// TwinCAT 3 PLC project mobject_collections
// Title: mobject-collections
// Company: mobject
// Author: mobject dev team
// ProjectVersion: 1.3.0
// ProgramVersion: 3.1.4023.0
// libraries:
//   Tc2_System, * (Beckhoff Automation GmbH)
//   Tc3_DynamicMemory, * (Beckhoff Automation GmbH)
//   mobject-disposable,1.1.1,mobject
//   mobject-enumerable,1.2.0,mobject
//   mobject-events,1.1.0,mobject
// project tree:
//   Dictionary/ Dictionary.TcPOU
//   Interfaces/Collections/Events/ I_CollectionChangedEvent.TcIO, I_CollectionDisposedEvent.TcIO (not stored)
//   Interfaces/Collections/ I_Collection.TcIO, I_List.TcIO, I_LinkedList.TcIO, I_Queue.TcIO, I_Stack.TcIO
//   Interfaces/Collections/Nodes/ I_CollectionNode.TcIO, I_LinkedListNode.TcIO, I_ListNode.TcIO
//   Interfaces/KeyValueCollections/Events/ I_KeyValueCollectionChangedEvent.TcIO, I_KeyValueCollectionDisposedEvent.TcIO
//   Interfaces/KeyValueCollections/ I_Dictionary.TcIO, I_KeyValueCollection.TcIO
//   Interfaces/KeyValueCollections/Nodes/ I_DictionaryTreeNode.TcIO, I_OrderedDictionaryTreeNode.TcIO
//   LinkedList/ LinkedList.TcPOU
//   List/ List.TcPOU
//   OrderedDictionary/ OrderedDictionary.TcPOU
//   Queue/ Queue.TcPOU
//   Stack/ Stack.TcPOU
//   _Internal/Dictionary/Enumerator/ DictionaryForwardEnumerator.TcPOU
//   _Internal/Dictionary/Node/ DictionaryTreeNode.TcPOU
//   _Internal/Events/Collection/ CollectionChangedEvent.TcPOU, CollectionDisposedEvent.TcPOU, CollectionEvent.TcPOU
//   _Internal/Events/KeyValueCollection/ KeyValueCollectionChangedEvent.TcPOU, KeyValueCollectionDisposedEvent.TcPOU, KeyValueCollectionEvent.TcPOU
//   _Internal/LinkedList/Enumerator/ LinkedListForwardEnumerator.TcPOU
//   _Internal/LinkedList/Node/ LinkedListNode.TcPOU
//   _Internal/List/Enumerator/ ListForwardEnumerator.TcPOU
//   _Internal/List/Node/ ListNode.TcPOU
//   _Internal/OrderedDictionary/Enumerator/ OrderedDictionaryForwardEnumerator.TcPOU
//   _Internal/OrderedDictionary/Node/ OrderedDictionaryTreeNode.TcPOU

// ---- Interfaces/Collections/Events/I_CollectionChangedEvent.TcIO
INTERFACE I_CollectionChangedEvent EXTENDS I_Event

PROPERTY PUBLIC Target : I_Collection
GET
END_GET
END_PROPERTY

END_INTERFACE

// ---- Interfaces/Collections/I_Collection.TcIO
INTERFACE I_Collection EXTENDS I_Enumerable, I_Disposable, I_EventEmitter

METHOD PUBLIC AddItem
VAR_INPUT
	Item : ANY;
END_VAR
END_METHOD

METHOD PUBLIC Clear
END_METHOD

METHOD PUBLIC Contains : BOOL;
VAR_INPUT
	Item : ANY;
END_VAR
END_METHOD

PROPERTY PUBLIC Count : DINT
GET
END_GET
END_PROPERTY

PROPERTY IsEmpty : BOOL
GET
END_GET
END_PROPERTY

METHOD PUBLIC TryCopyTo : BOOL
VAR_INPUT
	Destination : ANY;
END_VAR
END_METHOD

METHOD PUBLIC TryCopyToLocation : BOOL
VAR_INPUT
	DestinationAddress : PVOID;
	DestinationSize : UDINT;
END_VAR
END_METHOD

METHOD PUBLIC TryRemoveItem : BOOL
VAR_INPUT
	Item : ANY;
END_VAR
END_METHOD

END_INTERFACE

// ---- Interfaces/Collections/I_List.TcIO
INTERFACE I_List EXTENDS I_Collection

PROPERTY PUBLIC Capacity : DINT
GET
END_GET
END_PROPERTY

METHOD PUBLIC GetIndexOf : DINT
VAR_INPUT
	Item : ANY;
END_VAR
END_METHOD

METHOD PUBLIC TrimExcess
END_METHOD

METHOD PUBLIC TryGetByIndex : BOOL
VAR_INPUT
	Index : DINT;
	Destination : ANY;
END_VAR
END_METHOD

METHOD PUBLIC TryGetToByIndex : BOOL
VAR_INPUT
	Index : DINT;
	DestinationAddress : PVOID;
	DestinationSize : UDINT;
END_VAR
END_METHOD

METHOD TryInsert : BOOL
VAR_INPUT
	Index : DINT;
	Item : ANY;
END_VAR
END_METHOD

METHOD TryRemoveAt : BOOL
VAR_INPUT
	Index : DINT;
END_VAR
END_METHOD

END_INTERFACE

// ---- Interfaces/Collections/I_LinkedList.TcIO
INTERFACE I_LinkedList EXTENDS I_Collection

METHOD PUBLIC AddAfter
VAR_INPUT
	After : I_LinkedListNode;
	Value : ANY;
END_VAR
END_METHOD

METHOD PUBLIC AddBefore
VAR_INPUT
	Before : I_LinkedListNode;
	Value : ANY;
END_VAR
END_METHOD

METHOD PUBLIC AddFirst
VAR_INPUT
	Value : ANY;
END_VAR
END_METHOD

METHOD PUBLIC AddLast
VAR_INPUT
	Value : ANY;
END_VAR
END_METHOD

METHOD PUBLIC Find : I_LinkedListNode
VAR_INPUT
	Value : ANY;
END_VAR
END_METHOD

METHOD PUBLIC FindLast : I_LinkedListNode
VAR_INPUT
	Value : ANY;
END_VAR
END_METHOD

PROPERTY PUBLIC First : I_LinkedListNode
GET
END_GET
END_PROPERTY

PROPERTY PUBLIC Last : I_LinkedListNode
GET
END_GET
END_PROPERTY

METHOD PUBLIC Remove
VAR_INPUT
	Value : ANY;
END_VAR
END_METHOD

METHOD PUBLIC RemoveFirst
END_METHOD

METHOD PUBLIC RemoveLast
END_METHOD

END_INTERFACE

// ---- Interfaces/Collections/I_Queue.TcIO
INTERFACE I_Queue EXTENDS I_Collection

METHOD PUBLIC Enqueue
VAR_INPUT
	Item : ANY;
END_VAR
END_METHOD

METHOD PUBLIC TryDequeue : BOOL;
VAR_INPUT
	Destination : ANY;
END_VAR
END_METHOD

METHOD PUBLIC TryPeek : BOOL;
VAR_INPUT
	Destination : ANY;
END_VAR
END_METHOD

END_INTERFACE

// ---- Interfaces/Collections/I_Stack.TcIO
INTERFACE I_Stack EXTENDS I_Collection, I_EventEmitter

METHOD PUBLIC Push
VAR_INPUT
	Item : ANY;
END_VAR
END_METHOD

METHOD PUBLIC TryPeek : BOOL;
VAR_INPUT
	Destination : ANY;
END_VAR
END_METHOD

METHOD PUBLIC TryPop : BOOL;
VAR_INPUT
	Destination : ANY;
END_VAR
END_METHOD

END_INTERFACE

// ---- Interfaces/Collections/Nodes/I_CollectionNode.TcIO
INTERFACE I_CollectionNode EXTENDS I_Disposable

PROPERTY PUBLIC DataSize : UDINT
GET
END_GET
END_PROPERTY

METHOD PUBLIC Equals : BOOL
VAR_INPUT
	Symbol : ANY;
END_VAR
END_METHOD

METHOD PUBLIC TryGet : BOOL;
VAR_INPUT
	Destination : ANY;
END_VAR
END_METHOD

METHOD PUBLIC TryGetTo : BOOL;
VAR_INPUT
	DestinationAddress : PVOID;
	DestinationSize : UDINT;
END_VAR
END_METHOD

END_INTERFACE

// ---- Interfaces/Collections/Nodes/I_LinkedListNode.TcIO
INTERFACE I_LinkedListNode EXTENDS I_CollectionNode

PROPERTY PUBLIC Next : I_LinkedListNode
GET
END_GET
SET
END_SET
END_PROPERTY

PROPERTY PUBLIC Previous : I_LinkedListNode
GET
END_GET
SET
END_SET
END_PROPERTY

END_INTERFACE

// ---- Interfaces/Collections/Nodes/I_ListNode.TcIO
INTERFACE I_ListNode EXTENDS I_CollectionNode;

END_INTERFACE

// ---- Interfaces/KeyValueCollections/Events/I_KeyValueCollectionChangedEvent.TcIO
INTERFACE I_KeyValueCollectionChangedEvent EXTENDS I_Event

PROPERTY PUBLIC Target : I_KeyValueCollection
GET
END_GET
END_PROPERTY

END_INTERFACE

// ---- Interfaces/KeyValueCollections/Events/I_KeyValueCollectionDisposedEvent.TcIO
INTERFACE I_KeyValueCollectionDisposedEvent EXTENDS I_Event

PROPERTY PUBLIC Target : I_KeyValueCollection
GET
END_GET
END_PROPERTY

END_INTERFACE

// ---- Interfaces/KeyValueCollections/I_Dictionary.TcIO
INTERFACE I_Dictionary EXTENDS I_KeyValueCollection

METHOD PUBLIC AddOrUpdate
VAR_INPUT
	Key : T_MAXSTRING;
	Value : ANY;
END_VAR
END_METHOD

METHOD PUBLIC Clear
VAR_INPUT
END_VAR
END_METHOD

METHOD PUBLIC ContainsKey : BOOL
VAR_INPUT
	Key : T_MAXSTRING;
END_VAR
END_METHOD

METHOD PUBLIC GetKeys : I_Collection
END_METHOD

PROPERTY IsEmpty : BOOL
GET
END_GET
END_PROPERTY

METHOD PUBLIC Remove
VAR_INPUT
	Key : T_MAXSTRING;
END_VAR
END_METHOD

METHOD PUBLIC TryAdd : BOOL
VAR_INPUT
	Key : T_MAXSTRING;
	Value : ANY;
END_VAR
END_METHOD

METHOD PUBLIC TryGetValue : BOOL
VAR_INPUT
	Key : T_MAXSTRING;
	Destination	: ANY;
END_VAR
END_METHOD

METHOD PUBLIC TryGetValueTo : BOOL
VAR_INPUT
	Key : T_MAXSTRING;
	DestinationAddress : PVOID;
	DestinationSize : UDINT;
END_VAR
END_METHOD

END_INTERFACE

// ---- Interfaces/KeyValueCollections/I_KeyValueCollection.TcIO
INTERFACE I_KeyValueCollection EXTENDS I_KeyValueEnumerable, I_Enumerable, I_Disposable, I_EventEmitter

END_INTERFACE

// ---- Interfaces/KeyValueCollections/Nodes/I_DictionaryTreeNode.TcIO
INTERFACE I_DictionaryTreeNode EXTENDS I_CollectionNode

METHOD PUBLIC Clone
VAR_INPUT
	Node : I_DictionaryTreeNode;
END_VAR
END_METHOD

PROPERTY PUBLIC Height : DINT
GET
END_GET
SET
END_SET
END_PROPERTY

PROPERTY PUBLIC Key : T_MAXSTRING
GET
END_GET
END_PROPERTY

PROPERTY PUBLIC Left : I_DictionaryTreeNode
GET
END_GET
SET
END_SET
END_PROPERTY

PROPERTY PUBLIC NodeBufferPointer : Pointer To Byte
GET
END_GET
END_PROPERTY

PROPERTY PUBLIC NodeBufferSize : UDINT
GET
END_GET
END_PROPERTY

METHOD Reinitialize
VAR_INPUT
	Key : T_MAXSTRING;
	Source : ANY;
END_VAR
END_METHOD

PROPERTY PUBLIC Right : I_DictionaryTreeNode
GET
END_GET
SET
END_SET
END_PROPERTY

END_INTERFACE

// ---- Interfaces/KeyValueCollections/Nodes/I_OrderedDictionaryTreeNode.TcIO
INTERFACE I_OrderedDictionaryTreeNode EXTENDS I_CollectionNode

METHOD PUBLIC Clone
VAR_INPUT
	Node : I_OrderedDictionaryTreeNode;
END_VAR
END_METHOD

PROPERTY PUBLIC Height : DINT
GET
END_GET
SET
END_SET
END_PROPERTY

PROPERTY PUBLIC Key : T_MAXSTRING
GET
END_GET
END_PROPERTY

PROPERTY PUBLIC Left : I_OrderedDictionaryTreeNode
GET
END_GET
SET
END_SET
END_PROPERTY

PROPERTY PUBLIC Next : I_OrderedDictionaryTreeNode
GET
END_GET
SET
END_SET
END_PROPERTY

PROPERTY PUBLIC NodeBufferPointer : Pointer To Byte
GET
END_GET
END_PROPERTY

PROPERTY PUBLIC NodeBufferSize : UDINT
GET
END_GET
END_PROPERTY

PROPERTY PUBLIC Previous : I_OrderedDictionaryTreeNode
GET
END_GET
SET
END_SET
END_PROPERTY

METHOD Reinitialize
VAR_INPUT
	Key : T_MAXSTRING;
	Source : ANY;
END_VAR
END_METHOD

PROPERTY PUBLIC Right : I_OrderedDictionaryTreeNode
GET
END_GET
SET
END_SET
END_PROPERTY

END_INTERFACE

// ---- Dictionary/Dictionary.TcPOU
{attribute 'linkalways'} 
{attribute 'no_explicit_call' := 'This FB is a CLASS and must be accessed using methods or properties'}
{attribute 'enable_dynamic_creation'}
FUNCTION_BLOCK Dictionary EXTENDS Disposable IMPLEMENTS I_Dictionary
VAR
	eventEmitter : EventEmitter;
	rootNode : I_DictionaryTreeNode;
END_VAR

METHOD PUBLIC AddOrUpdate
VAR_INPUT
	Key : T_MAXSTRING;
	Value : ANY;
END_VAR
rootNode := THIS^.RecursiveInsert(Key, Value, rootNode);
EmitChangedEvent();
END_METHOD

METHOD PRIVATE Balance : I_DictionaryTreeNode
VAR_INPUT
	Node : I_DictionaryTreeNode;
END_VAR
VAR
	balanceFactor : DINT;
END_VAR
balanceFactor := THIS^.GetBalanceFactor(Node);

IF (balanceFactor > 1) THEN
	IF THIS^.GetBalanceFactor(Node.Left) < 0 THEN
		Node.Left := THIS^.LeftRotate(Node.Left);
	END_IF
	Node := RightRotate(Node);
ELSIF (balanceFactor < -1) THEN
	IF THIS^.GetBalanceFactor(Node.Right) > 0 THEN
		Node.Right := RightRotate(Node.Right);
	END_IF
	Node := LeftRotate(Node);
END_IF

Balance := Node;
END_METHOD

METHOD PUBLIC Clear
VAR_INPUT
END_VAR
IF rootNode = 0 THEN
	RETURN;
END_IF

THIS^.RecursiveClear(rootNode);
rootNode := 0;
EmitChangedEvent();
END_METHOD

METHOD PUBLIC ContainsKey : BOOL
VAR_INPUT
	Key : T_MAXSTRING;
END_VAR
VAR
	foundNode : I_DictionaryTreeNode;
END_VAR
foundNode := THIS^.RecursiveFind(Key, rootNode);

IF foundNode = 0 THEN
	RETURN;
END_IF

ContainsKey := TRUE;
END_METHOD

PROPERTY PUBLIC Count : DINT
GET
VAR
	NodeCount : DINT;
END_VAR
RecursiveCountNodes(rootNode, NodeCount);
Count := NodeCount;
END_GET
END_PROPERTY

METHOD PRIVATE EmitChangedEvent
VAR
	pDictionaryChangedEvent : POINTER TO KeyValueCollectionChangedEvent;
END_VAR
pDictionaryChangedEvent := __NEW(KeyValueCollectionChangedEvent(Target := THIS^));
eventEmitter.Emit('OnChanged', pDictionaryChangedEvent^);
pDictionaryChangedEvent^.Dispose();
END_METHOD

METHOD PRIVATE EmitDisposedEvent
VAR
	pDictionaryDisposedEvent : POINTER TO KeyValueCollectionDisposedEvent;
END_VAR
pDictionaryDisposedEvent := __NEW(KeyValueCollectionDisposedEvent(Target := THIS^));
eventEmitter.Emit('OnDisposed', pDictionaryDisposedEvent^);
pDictionaryDisposedEvent^.Dispose();
END_METHOD

METHOD FB_exit : BOOL
VAR_INPUT
	bInCopyCode : BOOL; // if TRUE, the exit method is called for exiting an instance that is copied afterwards (online change).
END_VAR
VAR
END_VAR
IF bInCopyCode THEN
    RETURN;
END_IF

Clear();
EmitDisposedEvent();
END_METHOD

METHOD PRIVATE FindMinimum : I_DictionaryTreeNode
VAR_INPUT
	Node : I_DictionaryTreeNode;
END_VAR
VAR
	nextNode : I_DictionaryTreeNode;
END_VAR
nextNode := Node;

WHILE (nextNode.left <> 0) DO
      nextNode := nextNode.left;
END_WHILE;

FindMinimum := nextNode;
END_METHOD

METHOD PRIVATE GetBalanceFactor : DINT
VAR_INPUT
	Node : I_DictionaryTreeNode;
END_VAR
IF (Node = 0) THEN
	GetBalanceFactor := 0;
	RETURN;
END_IF

GetBalanceFactor := THIS^.GetHeight(node.left) - THIS^.GetHeight(node.right);
END_METHOD

METHOD GetEnumerator : I_ForwardEnumerator
VAR
	pNodeCollection : POINTER TO LinkedList;
	pEnumerator : POINTER TO DictionaryForwardEnumerator;
END_VAR
pNodeCollection := __NEW(LinkedList);
THIS^.RecursiveAddNodesInOrderToCollection(rootNode, pNodeCollection^);

pEnumerator := __NEW(DictionaryForwardEnumerator(Parent := THIS^, Nodes := pNodeCollection^));
GetEnumerator := pEnumerator^;
END_METHOD

METHOD PRIVATE GetHeight : DINT
VAR_INPUT
	Node : I_DictionaryTreeNode;
END_VAR
IF Node = 0 THEN
	GetHeight := -1;
	RETURN;
END_IF

GetHeight := Node.Height;
END_METHOD

METHOD PUBLIC GetKeys : I_Collection
VAR
	pLinkedList : POINTER TO LinkedList;
END_VAR
pLinkedList := __NEW(LinkedList);
THIS^.RecursiveAddKeysInOrderToCollection(rootNode,pLinkedList^);
GetKeys := pLinkedList^;
END_METHOD

METHOD GetKeyValueEnumerator : I_KeyValueForwardEnumerator
VAR
	pNodeCollection : POINTER TO LinkedList;
	pEnumerator : POINTER TO DictionaryForwardEnumerator;
END_VAR
pNodeCollection := __NEW(LinkedList);
THIS^.RecursiveAddNodesInOrderToCollection(rootNode, pNodeCollection^);

pEnumerator := __NEW(DictionaryForwardEnumerator(Parent := THIS^, Nodes := pNodeCollection^));
GetKeyValueEnumerator := pEnumerator^;
END_METHOD

METHOD PRIVATE LeftRotate : I_DictionaryTreeNode
VAR_INPUT
	X : I_DictionaryTreeNode;
END_VAR
VAR
	y : I_DictionaryTreeNode;
	t2 : I_DictionaryTreeNode;
END_VAR
y := X.right;
t2 := y.left;
y.left := X;
X.right := t2;
THIS^.UpdateHeight(X);
THIS^.UpdateHeight(y);
LeftRotate := y;
END_METHOD

METHOD PUBLIC OffEvent
VAR_INPUT
	EventName : T_MaxString;
	EventHandler : I_EventHandler;
END_VAR
eventEmitter.OffEvent(EventName, EventHandler);
END_METHOD

METHOD PUBLIC OnceEvent
VAR_INPUT
	EventName : T_MaxString;
	EventHandler : I_EventHandler;
END_VAR
eventEmitter.OnceEvent(EventName, EventHandler);
END_METHOD

METHOD PUBLIC OnEvent
VAR_INPUT
	EventName : T_MaxString;
	EventHandler : I_EventHandler;
END_VAR
eventEmitter.OnEvent(EventName, EventHandler);
END_METHOD

METHOD PRIVATE RecursiveAddKeysInOrderToCollection
VAR_INPUT
	Node : I_DictionaryTreeNode;
	Collection : I_Collection;
END_VAR
VAR
	key : T_MAXSTRING;
END_VAR
IF Node = 0 THEN
	RETURN;
END_IF

THIS^.RecursiveAddKeysInOrderToCollection(Node.Left,Collection);
key := Node.Key;
Collection.AddItem(key);
THIS^.RecursiveAddKeysInOrderToCollection(Node.Right,Collection);
END_METHOD

METHOD PRIVATE RecursiveAddNodesInOrderToCollection
VAR_INPUT
	Node : I_DictionaryTreeNode;
	Collection : I_Collection;
END_VAR
IF Node = 0 THEN
	RETURN;
END_IF

THIS^.RecursiveAddNodesInOrderToCollection(Node.Left,Collection);
Collection.AddItem(Node);
THIS^.RecursiveAddNodesInOrderToCollection(Node.Right,Collection);
END_METHOD

METHOD PRIVATE RecursiveClear
VAR_INPUT
	Node : I_DictionaryTreeNode;
END_VAR
VAR
	thisNodeKey : T_MAXSTRING;
	leftNodeKey : T_MAXSTRING;
	rightNodeKey : T_MAXSTRING;
END_VAR
IF (Node = 0) THEN
	RETURN;
END_IF

thisNodeKey := Node.key;

IF (Node.Left <> 0) THEN
	leftNodeKey := Node.Left.key;
END_IF

IF (Node.Right <> 0) THEN
	rightNodeKey := Node.Right.key;
END_IF


RecursiveClear(Node.Left);
RecursiveClear(Node.Right);
Node.Dispose();
END_METHOD

METHOD PRIVATE RecursiveCountNodes
VAR_INPUT
	Node : I_DictionaryTreeNode;
	Count : REFERENCE TO DINT;
END_VAR
IF Node = 0 THEN
	RETURN;
END_IF

Count := Count + 1;

THIS^.RecursiveCountNodes(Node.Left,Count);
THIS^.RecursiveCountNodes(Node.Right,Count);
END_METHOD

METHOD PRIVATE RecursiveDelete : I_DictionaryTreeNode
VAR_INPUT
	Key : T_MAXSTRING;
	Node : I_DictionaryTreeNode;
END_VAR
VAR
	newNode : I_DictionaryTreeNode; 
	minValueNode : I_DictionaryTreeNode;
	minValueNodeParent : I_DictionaryTreeNode;
	balanceFactor : DINT;
END_VAR
IF (Node = 0) THEN
    RETURN;
END_IF

IF (Key < Node.Key) THEN
    Node.left := THIS^.RecursiveDelete(Key, Node.left);
ELSIF (Key > Node.Key) THEN
    Node.right := THIS^.RecursiveDelete(Key, Node.right);
ELSE
    IF (Node.Left = 0) OR (Node.Right = 0) THEN
        IF (Node.Left = 0) THEN
            newNode := Node.Right;
        ELSE
            newNode := Node.Left;
        END_IF

        Node.Dispose();
        THIS^.updateHeight(newNode);
        RecursiveDelete := THIS^.Balance(newNode);
        RETURN;
    ELSE
        minValueNode := FindMinimum(Node.Right);
        Node.Clone(minValueNode);
        Node.Right := THIS^.RecursiveDelete(minValueNode.Key, Node.Right);	
    END_IF
END_IF

THIS^.updateHeight(Node);
RecursiveDelete := THIS^.Balance(Node);
END_METHOD

METHOD PRIVATE RecursiveFind : I_DictionaryTreeNode
VAR_INPUT
	Key : T_MAXSTRING;
	Node : I_DictionaryTreeNode;
END_VAR
IF (Node = 0) THEN
	RETURN;
END_IF

IF (Key < Node.key) THEN
  RecursiveFind := THIS^.RecursiveFind(key, Node.left);
  RETURN;
ELSIF (key > Node.key) THEN
  RecursiveFind := THIS^.RecursiveFind(key, Node.right);
  RETURN;
ELSE 
  RecursiveFind := Node;
  RETURN;
END_IF
END_METHOD

METHOD PRIVATE RecursiveInsert : I_DictionaryTreeNode
VAR_INPUT
	Key : T_MAXSTRING;
	Value : ANY;
	Node : I_DictionaryTreeNode;
END_VAR
VAR
	pAVLTreeNode : POINTER TO DictionaryTreeNode;
	balanceFactor : DINT;
END_VAR
IF (Node = 0) THEN
	pAVLTreeNode := __NEW(DictionaryTreeNode(NodeKey := Key, NodeSource := Value));
	RecursiveInsert := pAVLTreeNode^;
	RETURN;
END_IF

IF (Key < Node.Key) THEN
	Node.left := THIS^.RecursiveInsert(Key, Value, Node.left);
ELSIF (Key > Node.Key) THEN
	Node.right := THIS^.RecursiveInsert(Key, Value, Node.right);
ELSE
	Node.Reinitialize(Key,Value);
	RecursiveInsert := Node;
END_IF

THIS^.updateHeight(node);

balanceFactor := THIS^.GetBalanceFactor(Node);
Node := balance(Node);
RecursiveInsert := Node;
END_METHOD

METHOD PUBLIC Remove
VAR_INPUT
	Key : T_MAXSTRING;
END_VAR
rootNode := THIS^.RecursiveDelete(Key, rootNode);
EmitChangedEvent();
END_METHOD

METHOD PRIVATE RightRotate : I_DictionaryTreeNode
VAR_INPUT
	Y : I_DictionaryTreeNode;
END_VAR
VAR
	x : I_DictionaryTreeNode;
	t2 : I_DictionaryTreeNode;
END_VAR
x := Y.left;
t2 := x.right;
x.right := Y;
Y.left := t2;
THIS^.UpdateHeight(Y);
THIS^.UpdateHeight(x);
RightRotate := x;
END_METHOD

METHOD PUBLIC TryAdd : BOOL
VAR_INPUT
	Key : T_MAXSTRING;
	Value : ANY;
END_VAR
IF ContainsKey(Key) THEN
	RETURN;
END_IF
	  
THIS^.AddOrUpdate(Key, Value);
TryAdd := TRUE;
END_METHOD

METHOD PUBLIC TryGetValue : BOOL
VAR_INPUT
	Key : T_MAXSTRING;
	Destination	: ANY;
END_VAR
TryGetValue := TryGetValueTo(Key, Destination.pValue, DINT_TO_UDINT(Destination.diSize));
END_METHOD

METHOD PUBLIC TryGetValueTo : BOOL
VAR_INPUT
	Key : T_MAXSTRING;
	DestinationAddress : PVOID;
	DestinationSize : UDINT;
END_VAR
VAR
	foundNode : I_DictionaryTreeNode;
END_VAR
foundNode := THIS^.RecursiveFind(Key, rootNode);

IF foundNode = 0 THEN
	RETURN;
END_IF

TryGetValueTo := foundNode.TryGetTo(DestinationAddress, DestinationSize);
END_METHOD

METHOD PRIVATE UpdateHeight
VAR_INPUT
	Node : I_DictionaryTreeNode;
END_VAR
IF (Node = 0) THEN
	RETURN;
END_IF

Node.height := 1 + MAX(THIS^.GetHeight(Node.left), THIS^.GetHeight(Node.right));
END_METHOD

END_FUNCTION_BLOCK

// ---- _Internal/Events/KeyValueCollection/KeyValueCollectionChangedEvent.TcPOU
{attribute 'linkalways'} 
{attribute 'no_explicit_call' := 'This FB is a CLASS and must be accessed using methods or properties'}
{attribute 'enable_dynamic_creation'}
FUNCTION_BLOCK KeyValueCollectionChangedEvent EXTENDS KeyValueCollectionEvent IMPLEMENTS I_KeyValueCollectionChangedEvent

END_FUNCTION_BLOCK

// ---- _Internal/Events/KeyValueCollection/KeyValueCollectionEvent.TcPOU
{attribute 'linkalways'} 
{attribute 'no_explicit_call' := 'This FB is a CLASS and must be accessed using methods or properties'}
{attribute 'enable_dynamic_creation'}
FUNCTION_BLOCK ABSTRACT KeyValueCollectionEvent EXTENDS Disposable
VAR
	_target : I_KeyValueCollection;
END_VAR

METHOD FB_init : BOOL
VAR_INPUT
	bInitRetains : BOOL; // if TRUE, the retain variables are initialized (warm start / cold start)
	bInCopyCode : BOOL;  // if TRUE, the instance afterwards gets moved into the copy code (online change)
	Target : I_KeyValueCollection;
END_VAR
This^._target := Target;
END_METHOD

PROPERTY PUBLIC Target : I_KeyValueCollection
GET // PUBLIC
Target := _target;
END_GET
END_PROPERTY

END_FUNCTION_BLOCK

// ---- _Internal/Events/KeyValueCollection/KeyValueCollectionDisposedEvent.TcPOU
{attribute 'linkalways'} 
{attribute 'no_explicit_call' := 'This FB is a CLASS and must be accessed using methods or properties'}
{attribute 'enable_dynamic_creation'}
FUNCTION_BLOCK KeyValueCollectionDisposedEvent EXTENDS KeyValueCollectionEvent IMPLEMENTS I_KeyValueCollectionDisposedEvent

END_FUNCTION_BLOCK

// ---- LinkedList/LinkedList.TcPOU
{attribute 'linkalways'} 
{attribute 'no_explicit_call' := 'This FB is a CLASS and must be accessed using methods or properties'}
{attribute 'enable_dynamic_creation'}
FUNCTION_BLOCK LinkedList EXTENDS Disposable IMPLEMENTS I_LinkedList
VAR
	head : I_LinkedListNode;
	tail : I_LinkedListNode;
	eventEmitter : EventEmitter;
END_VAR

METHOD PUBLIC AddAfter
VAR_INPUT
	After : I_LinkedListNode;
	Value : ANY;
END_VAR
VAR
	node : I_LinkedListNode;
END_VAR
IF NOT ContainsLinkedListNode(After) THEN
	RETURN;
END_IF

node := CreateNode(Value);
AddNodeAfter(After,node);
EmitChangedEvent();
END_METHOD

METHOD PUBLIC AddBefore
VAR_INPUT
	Before : I_LinkedListNode;
	Value : ANY;
END_VAR
VAR
	node : I_LinkedListNode;
END_VAR
IF NOT ContainsLinkedListNode(Before) THEN
	RETURN;
END_IF

node := CreateNode(Value);
AddNodeBefore(Before,node);
EmitChangedEvent();
END_METHOD

METHOD PUBLIC AddFirst
VAR_INPUT
	Value : ANY;
END_VAR
VAR
	node : I_LinkedListNode;
END_VAR
node := CreateNode(Value);
AddNodeFirst(node);
EmitChangedEvent();
END_METHOD

METHOD PUBLIC AddItem
VAR_INPUT
	Item : ANY;
END_VAR
AddLast(Item);
END_METHOD

METHOD PUBLIC AddLast
VAR_INPUT
	Value : ANY;
END_VAR
VAR
	node : I_LinkedListNode;
END_VAR
node := CreateNode(Value);
AddNodeLast(node);
EmitChangedEvent();
END_METHOD

METHOD PRIVATE AddNodeAfter
VAR_INPUT
	After : I_LinkedListNode;
	Node : I_LinkedListNode;
END_VAR
VAR
	originalNext : I_LinkedListNode;
END_VAR
IF After = tail THEN
	AddNodeLast(Node);
	RETURN;
END_IF

originalNext := After.Next;
After.Next := Node;
Node.Previous := After;
Node.Next := originalNext;
originalNext.Previous := Node;
END_METHOD

METHOD PRIVATE AddNodeBefore
VAR_INPUT
	Before : I_LinkedListNode;
	Node : I_LinkedListNode;
END_VAR
VAR
	originalBefore : I_LinkedListNode;
END_VAR
IF Before = head THEN
	AddNodeFirst(Node);
	RETURN;
END_IF

originalBefore := Before.Previous;
Before.Previous := Node;
Node.Next := Before;
Node.Previous := originalBefore;
originalBefore.Next := Node;
END_METHOD

METHOD PRIVATE AddNodeFirst
VAR_INPUT
	Node : I_LinkedListNode;
END_VAR
VAR
	originalFirst : I_LinkedListNode;
END_VAR
IF IsEmpty THEN
	head := Node;
	tail := Node; 
	RETURN;	
END_IF

originalFirst := head;
head := Node;
Node.Next := originalFirst;
originalFirst.Previous := Node;
END_METHOD

METHOD PRIVATE AddNodeLast
VAR_INPUT
	Node : I_LinkedListNode;
END_VAR
VAR
	originalLast : I_LinkedListNode;
END_VAR
IF IsEmpty THEN
	head := Node;
	tail := Node; 
	RETURN;	
END_IF

originalLast := tail;
tail := Node;
Node.Previous := originalLast;
originalLast.Next := Node;
END_METHOD

METHOD PUBLIC Clear
IF IsEmpty THEN
	return;
END_IF

RemoveAllNodes();
EmitChangedEvent();
END_METHOD

METHOD PUBLIC Contains : BOOL
VAR_INPUT
    Item : ANY;
END_VAR
VAR
    found : I_LinkedListNode;
END_VAR
found := Find(Item);
Contains := found <> 0;
END_METHOD

METHOD PRIVATE ContainsLinkedListNode : BOOL
VAR_INPUT
    Node : I_LinkedListNode;
END_VAR
VAR
	current : I_LinkedListNode;
END_VAR
IF IsEmpty THEN	
	RETURN;
END_IF

current := head; 

WHILE current <> 0 DO
	IF current = Node THEN
		ContainsLinkedListNode := TRUE;
		RETURN;
	END_IF
	current := current.next; 
END_WHILE;
END_METHOD

PROPERTY PUBLIC Count : DINT
GET
VAR
	current : I_LinkedListNode;
END_VAR
current := First;

WHILE current <> 0 DO
	Count := Count + 1;
	current := current.Next;
END_WHILE
END_GET
END_PROPERTY

METHOD PRIVATE CreateNode : I_LinkedListNode
VAR_INPUT
	Value : ANY;
END_VAR
VAR
	pLinkedListItem : POINTER TO LinkedListNode;
END_VAR
pLinkedListItem := __NEW(LinkedListNode(Source := Value)); 
CreateNode := pLinkedListItem^;
END_METHOD

METHOD PRIVATE EmitChangedEvent
VAR
	pCollectionChangedEvent : POINTER TO CollectionChangedEvent;
END_VAR
pCollectionChangedEvent := __NEW(CollectionChangedEvent(Target := THIS^));
eventEmitter.Emit('OnChanged', pCollectionChangedEvent^);
pCollectionChangedEvent^.Dispose();
END_METHOD

METHOD PRIVATE EmitDisposedEvent
VAR
	pCollectionDisposedEvent : POINTER TO CollectionDisposedEvent;
END_VAR
pCollectionDisposedEvent := __NEW(CollectionDisposedEvent(Target := THIS^));
eventEmitter.Emit('OnDisposed', pCollectionDisposedEvent^);
pCollectionDisposedEvent^.Dispose();
END_METHOD

METHOD FB_exit : BOOL
VAR_INPUT
	bInCopyCode : BOOL; // if TRUE, the exit method is called for exiting an instance that is copied afterwards (online change).
END_VAR
IF bInCopyCode THEN
	RETURN;
END_IF

Clear();
EmitDisposedEvent();
END_METHOD

METHOD PUBLIC Find : I_LinkedListNode
VAR_INPUT
	Value : ANY;
END_VAR
Find := FindFirstNodeWithValue(Value);
END_METHOD

METHOD PRIVATE FindFirstNodeWithValue : I_LinkedListNode
VAR_INPUT
	Value : ANY;
END_VAR
VAR
	current : I_LinkedListNode;
END_VAR
IF IsEmpty THEN	
	RETURN;
END_IF

current := head; 

WHILE current <> 0 DO
	IF current.Equals(Value) THEN
		FindFirstNodeWithValue := current;
		RETURN;
	END_IF
	current := current.next; 
END_WHILE;
END_METHOD

METHOD PUBLIC FindLast : I_LinkedListNode
VAR_INPUT
	Value : ANY;
END_VAR
FindLast := FindLastNodeWithValue(Value);
END_METHOD

METHOD PRIVATE FindLastNodeWithValue : I_LinkedListNode
VAR_INPUT
	Value : ANY;
END_VAR
VAR
	current : I_LinkedListNode;
END_VAR
IF IsEmpty THEN	
	RETURN;
END_IF

current := tail; 

WHILE current <> 0 DO
	IF current.Equals(Value) THEN
		FindLastNodeWithValue := current;
		RETURN;
	END_IF
	current := current.Previous; 
END_WHILE;
END_METHOD

PROPERTY PUBLIC First : I_LinkedListNode
GET
First := head;
END_GET
END_PROPERTY

METHOD PUBLIC GetEnumerator : I_ForwardEnumerator
VAR
	pLinkedListForwardEnumerator : POINTER TO LinkedListForwardEnumerator;
END_VAR
pLinkedListForwardEnumerator := __NEW(LinkedListForwardEnumerator(Parent := THIS^));
GetEnumerator := pLinkedListForwardEnumerator^;
END_METHOD

PROPERTY IsEmpty : BOOL
GET
IsEmpty := head = 0;
END_GET
END_PROPERTY

PROPERTY PUBLIC Last : I_LinkedListNode
GET
Last := tail;
END_GET
END_PROPERTY

METHOD PUBLIC OffEvent
VAR_INPUT
	EventName : T_MaxString;
	EventHandler : I_EventHandler;
END_VAR
eventEmitter.OffEvent(EventName, EventHandler);
END_METHOD

METHOD PUBLIC OnceEvent
VAR_INPUT
	EventName : T_MaxString;
	EventHandler : I_EventHandler;
END_VAR
eventEmitter.OnceEvent(EventName, EventHandler);
END_METHOD

METHOD PUBLIC OnEvent
VAR_INPUT
	EventName : T_MaxString;
	EventHandler : I_EventHandler;
END_VAR
eventEmitter.OnEvent(EventName, EventHandler);
END_METHOD

METHOD PUBLIC Remove
VAR_INPUT
	Value : ANY;
END_VAR
TryRemoveItem(Value);
END_METHOD

METHOD PRIVATE RemoveAllNodes
WHILE First <> 0 DO
	RemoveNode(First);
END_WHILE
END_METHOD

METHOD PUBLIC RemoveFirst
IF IsEmpty THEN
	RETURN;
END_IF

RemoveNode(First);
EmitChangedEvent();
END_METHOD

METHOD PUBLIC RemoveLast
IF IsEmpty THEN
	RETURN;
END_IF

RemoveNode(Last);
EmitChangedEvent();
END_METHOD

METHOD PRIVATE RemoveNode : BOOL
VAR_INPUT
	Node : I_LinkedListNode;
END_VAR
IF IsEmpty THEN
	RETURN;
END_IF

IF Node = head AND Node = tail THEN
	// node is the only node
	head := 0;
	tail := 0;
	Node.Dispose();
	RETURN;
	
ELSIF Node = head THEN
	// node is the head
	head := node.Next;
	head.Previous := 0;	
	Node.Dispose();
	RETURN;
	
ELSIF Node = tail THEN
	// node is the tail
	tail := node.Previous;
	tail.Next := 0;	
	Node.Dispose();
	RETURN;
ELSE 
	// node is in the middle
	Node.Previous.Next := Node.Next;
	Node.Next.Previous := Node.Previous;
	Node.Dispose();
	RETURN;
END_IF
END_METHOD

METHOD PUBLIC TryCopyTo : BOOL
VAR_INPUT
	Destination : ANY;
END_VAR
TryCopyTo := TryCopyToLocation(Destination.pValue, DINT_TO_UDINT(Destination.diSize));
END_METHOD

METHOD PUBLIC TryCopyToLocation : BOOL
VAR_INPUT
	DestinationAddress : PVOID;
	DestinationSize : UDINT;
END_VAR
VAR
	currentNode : I_LinkedListNode;
	requiredDestinationSize : UDINT;
	currentPointer : pvoid;
END_VAR
currentNode := First;

// first pass we check to see what the total size of the list will be.
WHILE currentNode <> 0 DO
	requiredDestinationSize := requiredDestinationSize + currentNode.DataSize;
	currentNode := currentNode.Next;
END_WHILE

// we will not process the copy if the destination is too small.
IF DestinationSize <> requiredDestinationSize THEN
	RETURN;
END_IF

currentPointer := DestinationAddress;
currentNode := First;

WHILE currentNode <> 0 DO
	currentNode.TryGetTo(currentPointer,currentNode.DataSize);
	currentPointer := currentPointer + currentNode.DataSize;
	currentNode := currentNode.Next;
END_WHILE
END_METHOD

METHOD PUBLIC TryRemoveItem : BOOL
VAR_INPUT
	Item : ANY;
END_VAR
VAR
	foundNode : I_LinkedListNode;
END_VAR
foundNode := FindFirstNodeWithValue(Item);

IF foundNode = 0 THEN
	RETURN;
END_IF

RemoveNode(foundNode);
EmitChangedEvent();

TryRemoveItem := TRUE;
END_METHOD

END_FUNCTION_BLOCK

// ---- _Internal/LinkedList/Node/LinkedListNode.TcPOU
{attribute 'linkalways'} 
{attribute 'no_explicit_call' := 'This FB is a CLASS and must be accessed using methods or properties'}
{attribute 'enable_dynamic_creation'}
FUNCTION_BLOCK LinkedListNode EXTENDS Disposable IMPLEMENTS I_LinkedListNode
VAR
	pBuffer : POINTER TO BYTE;
	bufferSize : UDINT;
	_previous : I_LinkedListNode;
	_next : I_LinkedListNode;
END_VAR

METHOD PRIVATE CopyBufferToDestination
VAR_INPUT
	DestinationAddress : PVOID;
END_VAR
MEMCPY(DestinationAddress, pBuffer, bufferSize);
END_METHOD

METHOD PRIVATE CopySourceToBuffer
VAR_INPUT
	SourceAddress : PVOID;
END_VAR
MEMCPY(pBuffer, SourceAddress, bufferSize);
END_METHOD

METHOD PRIVATE CreateBuffer
VAR_INPUT
	SizeInBytes : UDINT;
END_VAR
bufferSize := SizeInBytes;
pBuffer := __NEW(BYTE, SizeInBytes);
END_METHOD

PROPERTY PUBLIC DataSize : UDINT
GET // PUBLIC
DataSize := bufferSize;
END_GET
END_PROPERTY

METHOD PRIVATE DestroyBuffer
IF pBuffer = 0 THEN
	RETURN;
END_IF

__DELETE(pBuffer);
bufferSize := 0;
END_METHOD

METHOD PUBLIC Equals : BOOL
VAR_INPUT
	Symbol : ANY;
END_VAR
IF pBuffer = 0 THEN
	RETURN;
END_IF

IF bufferSize <> DINT_TO_UDINT(Symbol.diSize) THEN
	RETURN;
END_IF

Equals := MEMCMP(Symbol.pValue, pBuffer, bufferSize) = 0;
END_METHOD

METHOD FB_exit : BOOL
VAR_INPUT
	bInCopyCode : BOOL; // if TRUE, the exit method is called for exiting an instance that is copied afterwards (online change).
END_VAR
IF bInCopyCode THEN
	RETURN;
END_IF

DestroyBuffer();
END_METHOD

METHOD FB_init : BOOL
VAR_INPUT
	bInitRetains : BOOL; // if TRUE, the retain variables are initialized (warm start / cold start)
	bInCopyCode : BOOL;  // if TRUE, the instance afterwards gets moved into the copy code (online change)
	Source : ANY;
END_VAR
CreateBuffer(DINT_TO_UDINT(Source.diSize));
CopySourceToBuffer(Source.pValue);
END_METHOD

PROPERTY PUBLIC Next : I_LinkedListNode
GET // PUBLIC
Next := _next;
END_GET
SET // PUBLIC
_next := Next;
END_SET
END_PROPERTY

PROPERTY PUBLIC Previous : I_LinkedListNode
GET // PUBLIC
Previous := _previous;
END_GET
SET // PUBLIC
_previous := Previous;
END_SET
END_PROPERTY

METHOD PUBLIC TryGet : BOOL;
VAR_INPUT
	Destination : ANY;
END_VAR
TryGet := TryGetTo(Destination.pValue, DINT_TO_UDINT(Destination.diSize));
END_METHOD

METHOD PUBLIC TryGetTo : BOOL;
VAR_INPUT
	DestinationAddress : PVOID;
	DestinationSize : UDINT;
END_VAR
IF pBuffer = 0 THEN
	RETURN;
END_IF

IF bufferSize <> DestinationSize THEN
	RETURN;
END_IF

CopyBufferToDestination(DestinationAddress);
TryGetTo := TRUE;
END_METHOD

END_FUNCTION_BLOCK

// ---- _Internal/Events/Collection/CollectionChangedEvent.TcPOU
{attribute 'linkalways'} 
{attribute 'no_explicit_call' := 'This FB is a CLASS and must be accessed using methods or properties'}
{attribute 'enable_dynamic_creation'}
FUNCTION_BLOCK CollectionChangedEvent EXTENDS CollectionEvent IMPLEMENTS I_CollectionChangedEvent

END_FUNCTION_BLOCK

// ---- _Internal/Events/Collection/CollectionEvent.TcPOU
{attribute 'linkalways'} 
{attribute 'no_explicit_call' := 'This FB is a CLASS and must be accessed using methods or properties'}
{attribute 'enable_dynamic_creation'}
FUNCTION_BLOCK ABSTRACT CollectionEvent EXTENDS Disposable
VAR
	_target : I_Collection;
END_VAR

METHOD FB_init : BOOL
VAR_INPUT
	bInitRetains : BOOL; // if TRUE, the retain variables are initialized (warm start / cold start)
	bInCopyCode : BOOL;  // if TRUE, the instance afterwards gets moved into the copy code (online change)
	Target : I_Collection;
END_VAR
This^._target := Target;
END_METHOD

PROPERTY PUBLIC Target : I_Collection
GET // PUBLIC
Target := _target;
END_GET
END_PROPERTY

END_FUNCTION_BLOCK

// ---- _Internal/Events/Collection/CollectionDisposedEvent.TcPOU
{attribute 'linkalways'} 
{attribute 'no_explicit_call' := 'This FB is a CLASS and must be accessed using methods or properties'}
{attribute 'enable_dynamic_creation'}
FUNCTION_BLOCK CollectionDisposedEvent EXTENDS CollectionEvent IMPLEMENTS I_CollectionDisposedEvent

END_FUNCTION_BLOCK

// ---- _Internal/LinkedList/Enumerator/LinkedListForwardEnumerator.TcPOU
{attribute 'linkalways'} 
{attribute 'no_explicit_call' := 'This FB is a CLASS and must be accessed using methods or properties'}
{attribute 'enable_dynamic_creation'}
FUNCTION_BLOCK LinkedListForwardEnumerator EXTENDS Disposable IMPLEMENTS I_ForwardEnumerator, I_EventHandler
VAR
	parent : I_LinkedList;
	currentNode : I_LinkedListNode;
	moveNextCalled : BOOL := FALSE;
	invalid : BOOL := FALSE; 
END_VAR

METHOD FB_exit : BOOL
VAR_INPUT
	bInCopyCode : BOOL; // if TRUE, the exit method is called for exiting an instance that is copied afterwards (online change).
END_VAR
IF bInCopyCode THEN
	RETURN;
END_IF

IF parent = 0 THEN
	RETURN;
END_IF

parent.OffEvent('OnChanged',THIS^);
parent.OffEvent('OnDisposed',THIS^);
END_METHOD

METHOD FB_init : BOOL
VAR_INPUT
	bInitRetains : BOOL; // if TRUE, the retain variables are initialized (warm start / cold start)
	bInCopyCode : BOOL;  // if TRUE, the instance afterwards gets moved into the copy code (online change)
	Parent : I_LinkedList;
END_VAR
Parent.OnEvent('OnChanged',THIS^);
Parent.OnEvent('OnDisposed',THIS^);
this^.parent := Parent;
END_METHOD

METHOD PUBLIC HandleEvent
VAR_INPUT
	Event : I_Event;
END_VAR
VAR
	changedEvent : I_CollectionChangedEvent;
	disposedEvent : I_CollectionDisposedEvent;
END_VAR
IF __QUERYINTERFACE(Event, changedEvent) THEN
	invalid := TRUE;
	currentNode := 0;
ELSIF __QUERYINTERFACE(Event, disposedEvent) THEN
	parent := 0;
	Dispose();
END_IF
END_METHOD

PROPERTY PUBLIC IsValid : BOOL
GET // PUBLIC
IsValid := (not invalid and parent <> 0);
END_GET
END_PROPERTY

METHOD PUBLIC MoveNext : BOOL
IF invalid THEN
	RETURN;
END_IF

IF NOT moveNextCalled THEN
	moveNextCalled := TRUE;	
	currentNode := parent.First;
	MoveNext := currentNode <> 0;
	RETURN;
END_IF

IF currentNode = 0 THEN
	RETURN;
END_IF

if currentNode.Next <> 0 then
	currentNode := currentNode.Next;
	MoveNext := TRUE;	
	RETURN;
END_IF
END_METHOD

METHOD Reset
VAR_INPUT
END_VAR
moveNextCalled := FALSE;
currentNode := 0;
END_METHOD

METHOD PUBLIC TryGet : BOOL;
VAR_INPUT
	Destination : ANY;
END_VAR
IF currentNode <> 0 THEN
	TryGet := currentNode.TryGet(Destination);
END_IF
END_METHOD

METHOD PUBLIC TryGetTo : BOOL;
VAR_INPUT
	DestinationAddress : PVOID;
	DestinationSize : UDINT;
END_VAR
IF currentNode <> 0 THEN
	TryGetTo := currentNode.TryGetTo(DestinationAddress,DestinationSize);
END_IF
END_METHOD

END_FUNCTION_BLOCK

// ---- _Internal/Dictionary/Enumerator/DictionaryForwardEnumerator.TcPOU
{attribute 'linkalways'} 
{attribute 'no_explicit_call' := 'This FB is a CLASS and must be accessed using methods or properties'}
{attribute 'enable_dynamic_creation'}
FUNCTION_BLOCK DictionaryForwardEnumerator EXTENDS Disposable IMPLEMENTS I_KeyValueForwardEnumerator, I_EventHandler
VAR
	parent : I_Dictionary;
	nodes : I_Collection;
	collectionEnumerator : I_ForwardEnumerator;
	currentNode : I_DictionaryTreeNode;
	moveNextCalled : BOOL := FALSE;
	invalid : BOOL := FALSE; 
END_VAR

METHOD FB_exit : BOOL
VAR_INPUT
	bInCopyCode : BOOL; // if TRUE, the exit method is called for exiting an instance that is copied afterwards (online change).
END_VAR
IF bInCopyCode THEN
	RETURN;
END_IF

collectionEnumerator.Dispose();
nodes.Dispose();

IF parent = 0 THEN
	RETURN;
END_IF

parent.OffEvent('OnChanged',THIS^);
parent.OffEvent('OnDisposed',THIS^);
END_METHOD

METHOD FB_init : BOOL
VAR_INPUT
	bInitRetains : BOOL; // if TRUE, the retain variables are initialized (warm start / cold start)
	bInCopyCode : BOOL;  // if TRUE, the instance afterwards gets moved into the copy code (online change)
	Parent : I_Dictionary;
	Nodes : I_Collection;
END_VAR
Parent.OnEvent('OnChanged',THIS^);
Parent.OnEvent('OnDisposed',THIS^);
THIS^.parent := Parent;
THIS^.nodes := Nodes;
THIS^.collectionEnumerator := Nodes.GetEnumerator();
END_METHOD

METHOD PUBLIC HandleEvent
VAR_INPUT
	Event : I_Event;
END_VAR
VAR
	changedEvent : I_KeyValueCollectionChangedEvent;
	disposedEvent : I_KeyValueCollectionDisposedEvent;
END_VAR
IF __QUERYINTERFACE(Event, changedEvent) THEN
	invalid := TRUE;
	currentNode := 0;
ELSIF __QUERYINTERFACE(Event, disposedEvent) THEN
	parent := 0;	
	Dispose();
END_IF
END_METHOD

PROPERTY PUBLIC IsValid : BOOL
GET // PUBLIC
IsValid := (not invalid and parent <> 0);
END_GET
END_PROPERTY

PROPERTY PUBLIC Key : T_MAXSTRING
GET
IF NOT IsValid THEN
	RETURN;
END_IF

IF currentNode = 0 THEN
	RETURN;
END_IF

Key := currentNode.Key;
END_GET
END_PROPERTY

METHOD PUBLIC MoveNext : BOOL
IF invalid THEN
	RETURN;
END_IF

IF collectionEnumerator.MoveNext() THEN
	collectionEnumerator.TryGet(currentNode);
	MoveNext := TRUE;
END_IF
END_METHOD

METHOD Reset
VAR_INPUT
END_VAR
moveNextCalled := FALSE;
collectionEnumerator.Reset();
END_METHOD

METHOD PUBLIC TryGet : BOOL;
VAR_INPUT
	Destination : ANY;
END_VAR
IF currentNode <> 0 THEN
	TryGet := currentNode.TryGet(Destination);
END_IF
END_METHOD

METHOD PUBLIC TryGetTo : BOOL;
VAR_INPUT
	DestinationAddress : PVOID;
	DestinationSize : UDINT;
END_VAR
IF currentNode <> 0 THEN
	TryGetTo := currentNode.TryGetTo(DestinationAddress,DestinationSize);
END_IF
END_METHOD

END_FUNCTION_BLOCK

// ---- _Internal/Dictionary/Node/DictionaryTreeNode.TcPOU
{attribute 'linkalways'} 
{attribute 'no_explicit_call' := 'This FB is a CLASS and must be accessed using methods or properties'}
{attribute 'enable_dynamic_creation'}
FUNCTION_BLOCK DictionaryTreeNode EXTENDS Disposable IMPLEMENTS I_DictionaryTreeNode
VAR
	_key : T_MAXSTRING;
	pBuffer : POINTER TO BYTE;
	bufferSize : UDINT;
    _height : DINT;
    _left : I_DictionaryTreeNode;
    _right : I_DictionaryTreeNode;
END_VAR

METHOD PUBLIC Clone
VAR_INPUT
	Node : I_DictionaryTreeNode;
END_VAR
DestroyBuffer();
CreateBuffer(Node.NodeBufferSize);
CopySourceToBuffer(Node.NodeBufferPointer);
_key := Node.Key;
END_METHOD

METHOD PRIVATE CopyBufferToDestination
VAR_INPUT
	DestinationAddress : PVOID;
END_VAR
MEMCPY(DestinationAddress, pBuffer, bufferSize);
END_METHOD

METHOD PRIVATE CopySourceToBuffer
VAR_INPUT
	SourceAddress : PVOID;
END_VAR
MEMCPY(pBuffer, SourceAddress, bufferSize);
END_METHOD

METHOD PRIVATE CreateBuffer
VAR_INPUT
	SizeInBytes : UDINT;
END_VAR
bufferSize := SizeInBytes;
pBuffer := __NEW(BYTE, SizeInBytes);
END_METHOD

PROPERTY PUBLIC DataSize : UDINT
GET
DataSize := bufferSize;
END_GET
END_PROPERTY

METHOD PRIVATE DestroyBuffer
VAR_INPUT
END_VAR
IF pBuffer = 0 THEN
	RETURN;
END_IF

__DELETE(pBuffer);
bufferSize := 0;
END_METHOD

METHOD PUBLIC Equals : BOOL
VAR_INPUT
	Symbol : ANY;
END_VAR
IF pBuffer = 0 THEN
	RETURN;
END_IF

IF bufferSize <> DINT_TO_UDINT(symbol.diSize) THEN
	RETURN;
END_IF

Equals := MEMCMP(Symbol.pValue, pBuffer, bufferSize) = 0;
END_METHOD

METHOD FB_exit : BOOL
VAR_INPUT
	bInCopyCode : BOOL; // if TRUE, the exit method is called for exiting an instance that is copied afterwards (online change).
END_VAR
IF bInCopyCode THEN
	RETURN;
END_IF

DestroyBuffer();
END_METHOD

METHOD FB_init : BOOL
VAR_INPUT
	bInitRetains : BOOL; // if TRUE, the retain variables are initialized (warm start / cold start)
	bInCopyCode : BOOL;  // if TRUE, the instance afterwards gets moved into the copy code (online change)
	NodeKey : T_MAXSTRING;
	NodeSource : ANY;
END_VAR
_key := NodeKey;
CreateBuffer(DINT_TO_UDINT(NodeSource.diSize));
CopySourceToBuffer(NodeSource.pValue);
END_METHOD

PROPERTY PUBLIC Height : DINT
GET
Height := _height;
END_GET
SET // PUBLIC
_height := Height;
END_SET
END_PROPERTY

PROPERTY PUBLIC Key : T_MAXSTRING
GET
Key := _key;
END_GET
END_PROPERTY

PROPERTY PUBLIC Left : I_DictionaryTreeNode
GET
Left := _left;
END_GET
SET
_left := Left;
END_SET
END_PROPERTY

PROPERTY PUBLIC NodeBufferPointer : Pointer To Byte
GET
NodeBufferPointer := pBuffer;
END_GET
END_PROPERTY

PROPERTY PUBLIC NodeBufferSize : UDINT
GET
NodeBufferSize := bufferSize;
END_GET
END_PROPERTY

METHOD Reinitialize
VAR_INPUT
	Key : T_MAXSTRING;
	Source : ANY;
END_VAR
_key := Key;

IF pBuffer <> 0 THEN
	DestroyBuffer();
END_IF

CreateBuffer(DINT_TO_UDINT(Source.diSize));
CopySourceToBuffer(Source.pValue);
END_METHOD

PROPERTY PUBLIC Right : I_DictionaryTreeNode
GET
Right := _right;
END_GET
SET
_right := Right;
END_SET
END_PROPERTY

METHOD TryGet : BOOL
VAR_INPUT
	Destination	: ANY;
END_VAR
TryGet := TryGetTo(Destination.pValue, DINT_TO_UDINT(Destination.diSize));
END_METHOD

METHOD TryGetTo : BOOL
VAR_INPUT
	DestinationAddress : PVOID;
	DestinationSize : UDINT;
END_VAR
IF pBuffer = 0 THEN
	RETURN;
END_IF

IF bufferSize <> DestinationSize THEN
	RETURN;
END_IF

CopyBufferToDestination(DestinationAddress);
TryGetTo := TRUE;
END_METHOD

END_FUNCTION_BLOCK

// ---- List/List.TcPOU
{attribute 'linkalways'} 
{attribute 'no_explicit_call' := 'This FB is a CLASS and must be accessed using methods or properties'}
{attribute 'enable_dynamic_creation'}
{attribute 'hide_all_locals'}
FUNCTION_BLOCK PUBLIC FINAL List EXTENDS Disposable IMPLEMENTS I_List
VAR
	memoryManager : FB_DynMem_Manager2;
	buffer : FB_DynMem_Buffer(ipMemMan := memoryManager);
	pArrayOfListNodes : POINTER TO I_ListNode;
	arrayCapacity : DINT;
	itemCount : DINT;
	eventEmitter : EventEmitter;
END_VAR

METHOD PUBLIC AddItem
VAR_INPUT
	Item : ANY;
END_VAR
VAR
	node : I_ListNode;
END_VAR
node := CreateNewNode(Item);
AddNodeLast(node);
EmitChangedEvent();
END_METHOD

METHOD PRIVATE AddNodeAt
VAR_INPUT
	Index : DINT;
	Node : I_ListNode;
END_VAR
VAR
	i : DINT;
END_VAR
IF Index = itemCount THEN
	AddNodeLast(Node);
	RETURN;
END_IF

IF Index > itemCount - 1 THEN
	RETURN;
END_IF

IF Count + 1 > arrayCapacity THEN
	Resize();
END_IF

//Move all excisting nodes up
FOR i := itemCount - 1 TO Index BY -1 DO
	pArrayOfListNodes[i + 1] := pArrayOfListNodes[i];
	pArrayOfListNodes[i] := 0;
END_FOR

pArrayOfListNodes[Index] := Node;
itemCount := itemCount + 1;
END_METHOD

METHOD PRIVATE AddNodeLast
VAR_INPUT
	Node : I_ListNode;
END_VAR
IF Count = arrayCapacity THEN
    Resize();
END_IF

pArrayOfListNodes[itemCount] := Node;
itemCount := itemCount + 1;
END_METHOD

PROPERTY PUBLIC Capacity : DINT
GET
Capacity := arrayCapacity;
END_GET
END_PROPERTY

METHOD Clear
VAR_INPUT
END_VAR
IF IsEmpty THEN
	RETURN;
END_IF

RemoveAllNodes();
EmitChangedEvent();
END_METHOD

METHOD Contains : BOOL
VAR_INPUT
	Item : ANY;
END_VAR
IF IsEmpty THEN
	RETURN;
END_IF

Contains := GetIndexOf(Item) > -1;
END_METHOD

PROPERTY PUBLIC Count : DINT
GET
Count := itemCount;
END_GET
END_PROPERTY

METHOD PRIVATE CreateNewNode : I_ListNode
VAR_INPUT
	Value : ANY;
END_VAR
VAR
	pNode : POINTER TO ListNode;
END_VAR
pNode := __NEW(ListNode(Source := Value));
CreateNewNode := pNode^;
END_METHOD

METHOD PRIVATE EmitChangedEvent
VAR
	pCollectionChangedEvent : POINTER TO CollectionChangedEvent;
END_VAR
pCollectionChangedEvent := __NEW(CollectionChangedEvent(Target := THIS^));
eventEmitter.Emit('OnChanged', pCollectionChangedEvent^);
pCollectionChangedEvent^.Dispose();
END_METHOD

METHOD PRIVATE EmitDisposedEvent
VAR
	pCollectionDisposedEvent : POINTER TO CollectionDisposedEvent;
END_VAR
pCollectionDisposedEvent := __NEW(CollectionDisposedEvent(Target := THIS^));
eventEmitter.Emit('OnDisposed', pCollectionDisposedEvent^);
pCollectionDisposedEvent^.Dispose();
END_METHOD

METHOD FB_exit : BOOL
VAR_INPUT
	bInCopyCode : BOOL; // if TRUE, the exit method is called for exiting an instance that is copied afterwards (online change).
END_VAR
VAR
END_VAR
IF bInCopyCode THEN
    RETURN;
END_IF

Clear();
buffer.DeleteBuffer();
EmitDisposedEvent();
END_METHOD

METHOD GetEnumerator : I_ForwardEnumerator
VAR
	pEnumerator : POINTER TO ListForwardEnumerator;
END_VAR
pEnumerator := __NEW(ListForwardEnumerator(Parent := THIS^));
GetEnumerator := pEnumerator^;
END_METHOD

METHOD PUBLIC GetIndexOf : DINT
VAR_INPUT
	Item : ANY;
END_VAR
VAR
	node : I_ListNode;
	i : DINT;
END_VAR
GetIndexOf := -1;

IF IsEmpty THEN
	RETURN;
END_IF

FOR i := 0 TO itemCount - 1 DO
	node := THIS^.Item(i);
	
	IF node.Equals(Item) THEN
		GetIndexOf := i;
		RETURN;
	END_IF
END_FOR
END_METHOD

PROPERTY IsEmpty : BOOL
GET
IsEmpty := itemCount = 0;
END_GET
END_PROPERTY

METHOD PRIVATE IsNotValidIndex : BOOL
VAR_INPUT
	Index : DINT;
END_VAR
IsNotValidIndex := not IsValidIndex(Index);
END_METHOD

METHOD PRIVATE IsValidIndex : BOOL
VAR_INPUT
	Index : DINT;
END_VAR
IF Index < 0 THEN
	RETURN;
END_IF

IF Index >= itemCount THEN
	RETURN;
END_IF

IsValidIndex := TRUE;
END_METHOD

METHOD PRIVATE Item : I_ListNode
VAR_INPUT
	Index : DINT;
END_VAR
IF IsNotValidIndex(Index) THEN
	RETURN;
END_IF

Item := pArrayOfListNodes[Index];
END_METHOD

METHOD PUBLIC OffEvent
VAR_INPUT
	EventName : T_MaxString;
	EventHandler : I_EventHandler;
END_VAR
eventEmitter.OffEvent(EventName, EventHandler);
END_METHOD

METHOD PUBLIC OnceEvent
VAR_INPUT
	EventName : T_MaxString;
	EventHandler : I_EventHandler;
END_VAR
eventEmitter.OnceEvent(EventName, EventHandler);
END_METHOD

METHOD PUBLIC OnEvent
VAR_INPUT
	EventName : T_MaxString;
	EventHandler : I_EventHandler;
END_VAR
eventEmitter.OnEvent(EventName, EventHandler);
END_METHOD

METHOD PRIVATE RemoveAllNodes
VAR
	i : DINT;
END_VAR
FOR i := 0 TO itemCount - 1 DO
	IF pArrayOfListNodes[i] <> 0 THEN
		pArrayOfListNodes[i].Dispose();
	END_IF
END_FOR

itemCount := 0;
END_METHOD

METHOD PRIVATE Resize
VAR
	node : I_ListNode;
END_VAR
VAR CONSTANT
	INITIAL_CAPACITY : DINT := 4;
END_VAR
IF arrayCapacity = 0 THEN
	arrayCapacity := INITIAL_CAPACITY;
ELSE
	arrayCapacity := arrayCapacity * 2;
END_IF

IF buffer.bAvailable THEN
	buffer.Resize(nSize := DINT_TO_UDINT(arrayCapacity) * SIZEOF(node), bPreserve := TRUE, bReset := FALSE);
ELSE
	buffer.CreateBuffer(nSize := DINT_TO_UDINT(arrayCapacity) * SIZEOF(node), bReset := TRUE);
END_IF

pArrayOfListNodes := buffer.pBuffer;
END_METHOD

METHOD PUBLIC TrimExcess
VAR
	node : I_ListNode;
END_VAR
IF arrayCapacity = 0 THEN
	RETURN;
END_IF

IF arrayCapacity = itemCount THEN
	RETURN;
END_IF

arrayCapacity := itemCount;
buffer.Resize(nSize := DINT_TO_UDINT(arrayCapacity) * SIZEOF(node), bPreserve := TRUE, bReset := FALSE);
END_METHOD

METHOD PUBLIC TryCopyTo : BOOL
VAR_INPUT
	Destination	: ANY;
END_VAR
TryCopyTo := TryCopyToLocation(Destination.pValue, DINT_TO_UDINT(Destination.diSize));
END_METHOD

METHOD PUBLIC TryCopyToLocation : BOOL
VAR_INPUT
	DestinationAddress : PVOID;
	DestinationSize : UDINT;
END_VAR
VAR
	i : DINT;
	requiredSize : UDINT;
	current : I_ListNode;
	pCurrent : PVOID;
END_VAR
IF IsEmpty THEN
    RETURN;
END_IF

//Compute required size
FOR i := 0 TO Count - 1 DO
    current := Item(i);
    requiredSize := requiredSize + current.DataSize;
END_FOR

//If destination size is to small abort
IF DestinationSize < requiredSize THEN
    RETURN;
END_IF

pCurrent := DestinationAddress;

FOR i := 0 TO Count - 1 DO
    current := Item(i);
    current.TryGetTo(pCurrent, current.DataSize);
    pCurrent := pCurrent + current.DataSize;
END_FOR
END_METHOD

METHOD PUBLIC TryGetByIndex : BOOL
VAR_INPUT
	Index : DINT;
	Destination : ANY;
END_VAR
VAR
	node : I_ListNode;
END_VAR
node := Item(Index);

IF node = 0 THEN
	RETURN;
END_IF

TryGetByIndex := node.TryGet(Destination);
END_METHOD

METHOD PUBLIC TryGetToByIndex : BOOL
VAR_INPUT
	Index : DINT;
	DestinationAddress : PVOID;
	DestinationSize : UDINT;
END_VAR
VAR
	node : I_ListNode;
END_VAR
node := Item(Index);

IF node = 0 THEN
	RETURN;
END_IF

TryGetToByIndex := node.TryGetTo(DestinationAddress, DestinationSize);
END_METHOD

METHOD TryInsert : BOOL
VAR_INPUT
	Index : DINT;
	Item : ANY;
END_VAR
VAR
	node : I_ListNode;
END_VAR
IF IsNotValidIndex(Index) THEN
	RETURN;
END_IF

node := CreateNewNode(Item);
AddNodeAt(Index, node);
EmitChangedEvent();
TryInsert := TRUE;
END_METHOD

METHOD PUBLIC TryRemoveAt : BOOL;
VAR_INPUT
	Index : DINT;
END_VAR
VAR
	i : DINT;
	node : I_ListNode;
END_VAR
IF IsNotValidIndex(Index) THEN
	RETURN;
END_IF

node := Item(Index);
node.Dispose();

FOR i := Index + 1 TO itemCount - 1 DO
	pArrayOfListNodes[i - 1] := pArrayOfListNodes[i];
	pArrayOfListNodes[i] := 0;
END_FOR

itemCount := itemCount - 1;
EmitChangedEvent();
TryRemoveAt := TRUE;
END_METHOD

METHOD TryRemoveItem : BOOL
VAR_INPUT
    Item : ANY;
END_VAR
VAR
    index : DINT;
END_VAR
index := GetIndexOf(Item);

IF index = -1 THEN
	RETURN;
END_IF

TryRemoveItem := TryRemoveAt(index);
END_METHOD

END_FUNCTION_BLOCK

// ---- _Internal/List/Node/ListNode.TcPOU
{attribute 'linkalways'} 
{attribute 'no_explicit_call' := 'This FB is a CLASS and must be accessed using methods or properties'}
{attribute 'enable_dynamic_creation'}
FUNCTION_BLOCK PUBLIC ListNode EXTENDS Disposable IMPLEMENTS I_ListNode
VAR
	pBuffer : POINTER TO BYTE;
	bufferSize : UDINT;
END_VAR

METHOD PRIVATE CopyBufferToDestination
VAR_INPUT
	DestinationAddress : PVOID;
END_VAR
MEMCPY(DestinationAddress, pBuffer, bufferSize);
END_METHOD

METHOD PRIVATE CopySourceToBuffer
VAR_INPUT
	SourceAddress : PVOID;
END_VAR
MEMCPY(pBuffer, SourceAddress, bufferSize);
END_METHOD

METHOD PRIVATE CreateBuffer
VAR_INPUT
	SizeInBytes : UDINT;
END_VAR
bufferSize := SizeInBytes;
pBuffer := __NEW(BYTE, SizeInBytes);
END_METHOD

PROPERTY PUBLIC DataSize : UDINT
GET
DataSize := bufferSize;
END_GET
END_PROPERTY

METHOD PRIVATE DestroyBuffer
VAR_INPUT
END_VAR
IF pBuffer = 0 THEN
	RETURN;
END_IF

__DELETE(pBuffer);
bufferSize := 0;
END_METHOD

METHOD PUBLIC Equals : BOOL
VAR_INPUT
	Symbol : ANY;
END_VAR
IF pBuffer = 0 THEN
	RETURN;
END_IF

IF bufferSize <> DINT_TO_UDINT(Symbol.diSize) THEN
	RETURN;
END_IF

Equals := memcmp(Symbol.pValue, pBuffer, bufferSize) = 0;
END_METHOD

METHOD FB_exit : BOOL
VAR_INPUT
	bInCopyCode : BOOL; // if TRUE, the exit method is called for exiting an instance that is copied afterwards (online change).
END_VAR
IF bInCopyCode THEN
	RETURN;
END_IF

DestroyBuffer();
END_METHOD

METHOD FB_init : BOOL
VAR_INPUT
	bInitRetains : BOOL; // if TRUE, the retain variables are initialized (warm start / cold start)
	bInCopyCode : BOOL;  // if TRUE, the instance afterwards gets moved into the copy code (online change)
	Source : ANY;
END_VAR
CreateBuffer(DINT_TO_UDINT(Source.diSize));
CopySourceToBuffer(Source.pValue);
END_METHOD

METHOD TryGet : BOOL
VAR_INPUT
	Destination	: ANY;
END_VAR
TryGet := TryGetTo(Destination.pValue, DINT_TO_UDINT(Destination.diSize));
END_METHOD

METHOD TryGetTo : BOOL
VAR_INPUT
	DestinationAddress : PVOID;
	DestinationSize : UDINT;
END_VAR
IF pBuffer = 0 THEN
	RETURN;
END_IF

IF bufferSize <> DestinationSize THEN
	RETURN;
END_IF

CopyBufferToDestination(DestinationAddress);
TryGetTo := TRUE;
END_METHOD

END_FUNCTION_BLOCK

// ---- _Internal/List/Enumerator/ListForwardEnumerator.TcPOU
{attribute 'no_explicit_call' := 'This FB is a CLASS and must be accessed using methods or properties'}
{attribute 'enable_dynamic_creation'}
FUNCTION_BLOCK ListForwardEnumerator EXTENDS Disposable IMPLEMENTS I_ForwardEnumerator, I_EventHandler
VAR
	parent : I_List;
	currentIndex : DINT := 0;
	invalid : BOOL := FALSE;
	moveNextCalled : BOOL := FALSE;
END_VAR

METHOD FB_exit : BOOL
VAR_INPUT
	bInCopyCode : BOOL; // if TRUE, the exit method is called for exiting an instance that is copied afterwards (online change).
END_VAR
IF bInCopyCode THEN
	RETURN;
END_IF

IF parent = 0 THEN
	RETURN;
END_IF

parent.OffEvent('OnChanged',THIS^);
parent.OffEvent('OnDisposed',THIS^);
END_METHOD

METHOD FB_init : BOOL
VAR_INPUT
	bInitRetains : BOOL; // if TRUE, the retain variables are initialized (warm start / cold start)
	bInCopyCode : BOOL;  // if TRUE, the instance afterwards gets moved into the copy code (online change)
	Parent : I_List;
END_VAR
Parent.OnEvent('OnChanged',THIS^);
Parent.OnEvent('OnDisposed',THIS^);
this^.parent := Parent;
END_METHOD

METHOD PUBLIC HandleEvent
VAR_INPUT
	Event : I_Event;
END_VAR
VAR
	changedEvent : I_CollectionChangedEvent;
	disposedEvent : I_CollectionDisposedEvent;
END_VAR
IF __QUERYINTERFACE(Event, changedEvent) THEN
	invalid := TRUE;
	currentIndex := 0;
ELSIF __QUERYINTERFACE(Event, disposedEvent) THEN
	parent := 0;
	Dispose();
END_IF
END_METHOD

PROPERTY PUBLIC IsValid : BOOL
GET
IsValid := (NOT invalid AND parent <> 0);
END_GET
END_PROPERTY

METHOD MoveNext : BOOL
IF invalid THEN
    RETURN;
END_IF

IF parent = 0 THEN
    RETURN;
END_IF

IF parent.Count = 0 THEN
    RETURN;
END_IF

IF NOT moveNextCalled THEN
	MoveNext := moveNextCalled := TRUE;
	RETURN;
END_IF

IF currentIndex < parent.Count - 1 THEN
    currentIndex := currentIndex + 1;
    MoveNext := TRUE;
END_IF
END_METHOD

METHOD Reset
VAR_INPUT
END_VAR
moveNextCalled := FALSE;
currentIndex := 0;
END_METHOD

METHOD PUBLIC TryGet : BOOL
VAR_INPUT
	Destination : ANY;
END_VAR
IF invalid THEN
	RETURN;
END_IF

IF parent = 0 THEN
	RETURN;
END_IF

IF NOT moveNextCalled THEN
	RETURN;
END_IF

TryGet := parent.TryGetByIndex(currentIndex, Destination);
END_METHOD

METHOD TryGetTo : BOOL
VAR_INPUT
	DestinationAddress : PVOID;
	DestinationSize : UDINT;
END_VAR
IF invalid THEN
	RETURN;
END_IF

IF parent = 0 THEN
	RETURN;
END_IF

IF NOT moveNextCalled THEN
	RETURN;
END_IF

TryGetTo := parent.TryGetToByIndex(currentIndex, DestinationAddress, DestinationSize);
END_METHOD

END_FUNCTION_BLOCK

// ---- OrderedDictionary/OrderedDictionary.TcPOU
{attribute 'linkalways'} 
{attribute 'no_explicit_call' := 'This FB is a CLASS and must be accessed using methods or properties'}
{attribute 'enable_dynamic_creation'}
FUNCTION_BLOCK OrderedDictionary EXTENDS Disposable IMPLEMENTS I_Dictionary
VAR
	eventEmitter : EventEmitter;
	rootNode : I_OrderedDictionaryTreeNode;
	head : I_OrderedDictionaryTreeNode;
	tail : I_OrderedDictionaryTreeNode;
END_VAR

METHOD PRIVATE AddKeysInOrderToCollection
VAR_INPUT
	Collection : I_Collection;
END_VAR
VAR
	currentNode : I_OrderedDictionaryTreeNode;
	key : T_MAXSTRING;
END_VAR
IF head = 0 THEN
	RETURN;
END_IF

currentNode := head;

REPEAT
    key := currentNode.Key;
	Collection.AddItem(key);
	currentNode := currentNode.Next;
UNTIL
    currentNode = 0
END_REPEAT;
END_METHOD

METHOD PRIVATE AddNodesInOrderToCollection
VAR_INPUT
	Collection : I_Collection;
END_VAR
VAR
	currentNode : I_OrderedDictionaryTreeNode;
	key : T_MAXSTRING;
END_VAR
IF head = 0 THEN
	RETURN;
END_IF

currentNode := head;

REPEAT
	Collection.AddItem(currentNode);
	currentNode := currentNode.Next;
UNTIL
    currentNode = 0
END_REPEAT;
END_METHOD

METHOD PRIVATE AddNodeToEnd
VAR_INPUT
	Node : I_OrderedDictionaryTreeNode;
END_VAR
IF head = 0 THEN
	head := Node;
	tail := Node;
	RETURN;
END_IF

Node.Previous := tail;
Node.Previous.Next := Node;
tail := Node;
END_METHOD

METHOD PUBLIC AddOrUpdate
VAR_INPUT
	Key : T_MAXSTRING;
	Value : ANY;
END_VAR
rootNode := THIS^.RecursiveInsert(Key, Value, rootNode);
EmitChangedEvent();
END_METHOD

METHOD PRIVATE Balance : I_OrderedDictionaryTreeNode
VAR_INPUT
	Node : I_OrderedDictionaryTreeNode;
END_VAR
VAR
	balanceFactor : DINT;
END_VAR
balanceFactor := THIS^.GetBalanceFactor(Node);

IF (balanceFactor > 1) THEN
	IF THIS^.GetBalanceFactor(Node.Left) < 0 THEN
		Node.Left := THIS^.LeftRotate(Node.Left);
	END_IF
	Node := RightRotate(Node);
ELSIF (balanceFactor < -1) THEN
	IF THIS^.GetBalanceFactor(Node.Right) > 0 THEN
		Node.Right := RightRotate(Node.Right);
	END_IF
	Node := LeftRotate(Node);
END_IF

Balance := Node;
END_METHOD

METHOD PUBLIC Clear
VAR_INPUT
END_VAR
IF rootNode = 0 THEN
	RETURN;
END_IF

THIS^.RecursiveClear(rootNode);
head := 0;
tail := 0;
rootNode := 0;
EmitChangedEvent();
END_METHOD

METHOD PUBLIC ContainsKey : BOOL
VAR_INPUT
	Key : T_MAXSTRING;
END_VAR
VAR
	foundNode : I_OrderedDictionaryTreeNode;
END_VAR
foundNode := THIS^.RecursiveFind(Key, rootNode);

IF foundNode = 0 THEN
	RETURN;
END_IF

ContainsKey := TRUE;
END_METHOD

PROPERTY PUBLIC Count : DINT
GET
VAR
	NodeCount : DINT;
END_VAR
RecursiveCountNodes(rootNode, NodeCount);
Count := NodeCount;
END_GET
END_PROPERTY

METHOD PRIVATE EmitChangedEvent
VAR
	pDictionaryChangedEvent : POINTER TO KeyValueCollectionChangedEvent;
END_VAR
pDictionaryChangedEvent := __NEW(KeyValueCollectionChangedEvent(Target := THIS^));
eventEmitter.Emit('OnChanged', pDictionaryChangedEvent^);
pDictionaryChangedEvent^.Dispose();
END_METHOD

METHOD PRIVATE EmitDisposedEvent
VAR
	pDictionaryDisposedEvent : POINTER TO KeyValueCollectionDisposedEvent;
END_VAR
pDictionaryDisposedEvent := __NEW(KeyValueCollectionDisposedEvent(Target := THIS^));
eventEmitter.Emit('OnDisposed', pDictionaryDisposedEvent^);
pDictionaryDisposedEvent^.Dispose();
END_METHOD

METHOD FB_exit : BOOL
VAR_INPUT
	bInCopyCode : BOOL; // if TRUE, the exit method is called for exiting an instance that is copied afterwards (online change).
END_VAR
VAR
END_VAR
IF bInCopyCode THEN
    RETURN;
END_IF

Clear();
EmitDisposedEvent();
END_METHOD

METHOD PRIVATE FindMinimum : I_OrderedDictionaryTreeNode
VAR_INPUT
	Node : I_OrderedDictionaryTreeNode;
END_VAR
VAR
	nextNode : I_OrderedDictionaryTreeNode;
END_VAR
nextNode := Node;

WHILE (nextNode.left <> 0) DO
      nextNode := nextNode.left;
END_WHILE;

FindMinimum := nextNode;
END_METHOD

METHOD PRIVATE GetBalanceFactor : DINT
VAR_INPUT
	Node : I_OrderedDictionaryTreeNode;
END_VAR
IF (Node = 0) THEN
	GetBalanceFactor := 0;
	RETURN;
END_IF

GetBalanceFactor := THIS^.GetHeight(node.left) - THIS^.GetHeight(node.right);
END_METHOD

METHOD GetEnumerator : I_ForwardEnumerator
VAR
	pNodeCollection : POINTER TO LinkedList;
	pEnumerator : POINTER TO OrderedDictionaryForwardEnumerator;
END_VAR
pNodeCollection := __NEW(LinkedList);
THIS^.AddNodesInOrderToCollection(pNodeCollection^);

pEnumerator := __NEW(OrderedDictionaryForwardEnumerator(Parent := THIS^, Nodes := pNodeCollection^));
GetEnumerator := pEnumerator^;
END_METHOD

METHOD PRIVATE GetHeight : DINT
VAR_INPUT
	Node : I_OrderedDictionaryTreeNode;
END_VAR
IF Node = 0 THEN
	GetHeight := -1;
	RETURN;
END_IF

GetHeight := Node.Height;
END_METHOD

METHOD PUBLIC GetKeys : I_Collection
VAR
	pLinkedList : POINTER TO LinkedList;
END_VAR
pLinkedList := __NEW(LinkedList);
THIS^.AddKeysInOrderToCollection(pLinkedList^);
GetKeys := pLinkedList^;
END_METHOD

METHOD GetKeyValueEnumerator : I_KeyValueForwardEnumerator
VAR
	pNodeCollection : POINTER TO LinkedList;
	pEnumerator : POINTER TO OrderedDictionaryForwardEnumerator;
END_VAR
pNodeCollection := __NEW(LinkedList);
THIS^.AddNodesInOrderToCollection(pNodeCollection^);

pEnumerator := __NEW(OrderedDictionaryForwardEnumerator(Parent := THIS^, Nodes := pNodeCollection^));
GetKeyValueEnumerator := pEnumerator^;
END_METHOD

PROPERTY IsEmpty : BOOL
GET
IsEmpty := rootNode = 0;
END_GET
END_PROPERTY

METHOD PRIVATE LeftRotate : I_OrderedDictionaryTreeNode
VAR_INPUT
	X : I_OrderedDictionaryTreeNode;
END_VAR
VAR
	y : I_OrderedDictionaryTreeNode;
	t2 : I_OrderedDictionaryTreeNode;
END_VAR
y := X.right;
t2 := y.left;
y.left := X;
X.right := t2;
THIS^.UpdateHeight(X);
THIS^.UpdateHeight(y);
LeftRotate := y;
END_METHOD

METHOD PUBLIC OffEvent
VAR_INPUT
	EventName : T_MaxString;
	EventHandler : I_EventHandler;
END_VAR
eventEmitter.OffEvent(EventName, EventHandler);
END_METHOD

METHOD PUBLIC OnceEvent
VAR_INPUT
	EventName : T_MaxString;
	EventHandler : I_EventHandler;
END_VAR
eventEmitter.OnceEvent(EventName, EventHandler);
END_METHOD

METHOD PUBLIC OnEvent
VAR_INPUT
	EventName : T_MaxString;
	EventHandler : I_EventHandler;
END_VAR
eventEmitter.OnEvent(EventName, EventHandler);
END_METHOD

METHOD PRIVATE RecursiveClear
VAR_INPUT
	Node : I_OrderedDictionaryTreeNode;
END_VAR
VAR
	thisNodeKey : T_MAXSTRING;
	leftNodeKey : T_MAXSTRING;
	rightNodeKey : T_MAXSTRING;
END_VAR
IF (Node = 0) THEN
	RETURN;
END_IF

thisNodeKey := Node.key;

IF (Node.Left <> 0) THEN
	leftNodeKey := Node.Left.key;
END_IF

IF (Node.Right <> 0) THEN
	rightNodeKey := Node.Right.key;
END_IF

RecursiveClear(Node.Left);
RecursiveClear(Node.Right);
Node.Dispose();
END_METHOD

METHOD PRIVATE RecursiveCountNodes
VAR_INPUT
	Node : I_OrderedDictionaryTreeNode;
	Count : REFERENCE TO DINT;
END_VAR
IF Node = 0 THEN
	RETURN;
END_IF

Count := Count + 1;

THIS^.RecursiveCountNodes(Node.Left,Count);
THIS^.RecursiveCountNodes(Node.Right,Count);
END_METHOD

METHOD PRIVATE RecursiveDelete : I_OrderedDictionaryTreeNode
VAR_INPUT
	Key : T_MAXSTRING;
	Node : I_OrderedDictionaryTreeNode;
END_VAR
VAR
	newNode : I_OrderedDictionaryTreeNode; 
	minValueNode : I_OrderedDictionaryTreeNode;
	minValueNodeParent : I_OrderedDictionaryTreeNode;
	balanceFactor : DINT;
END_VAR
IF (Node = 0) THEN
    RETURN;
END_IF

IF (Key < Node.Key) THEN
    Node.left := THIS^.RecursiveDelete(Key, Node.left);
ELSIF (Key > Node.Key) THEN
    Node.right := THIS^.RecursiveDelete(Key, Node.right);
ELSE
    IF (Node.Left = 0) OR (Node.Right = 0) THEN
        IF (Node.Left = 0) THEN
            newNode := Node.Right;
        ELSE
            newNode := Node.Left;
        END_IF
		RemoveNode(Node);
        Node.Dispose();
        THIS^.updateHeight(newNode);
        RecursiveDelete := THIS^.Balance(newNode);
        RETURN;
    ELSE
        minValueNode := FindMinimum(Node.Right);
        Node.Clone(minValueNode);
		ReplaceClonedNodeInOrder(Node, minValueNode);
        Node.Right := THIS^.RecursiveDelete(minValueNode.Key, Node.Right);	
    END_IF
END_IF

THIS^.updateHeight(Node);
RecursiveDelete := THIS^.Balance(Node);
END_METHOD

METHOD PRIVATE RecursiveFind : I_OrderedDictionaryTreeNode
VAR_INPUT
	Key : T_MAXSTRING;
	Node : I_OrderedDictionaryTreeNode;
END_VAR
IF (Node = 0) THEN
	RETURN;
END_IF

IF (Key < Node.key) THEN
  RecursiveFind := THIS^.RecursiveFind(key, Node.left);
  RETURN;
ELSIF (key > Node.key) THEN
  RecursiveFind := THIS^.RecursiveFind(key, Node.right);
  RETURN;
ELSE 
  RecursiveFind := Node;
  RETURN;
END_IF
END_METHOD

METHOD PRIVATE RecursiveInsert : I_OrderedDictionaryTreeNode
VAR_INPUT
	Key : T_MAXSTRING;
	Value : ANY;
	Node : I_OrderedDictionaryTreeNode;
END_VAR
VAR
	pAVLTreeNode : POINTER TO OrderedDictionaryTreeNode;
	balanceFactor : DINT;
END_VAR
IF (Node = 0) THEN
	pAVLTreeNode := __NEW(OrderedDictionaryTreeNode(NodeKey := Key, NodeSource := Value));
	AddNodeToEnd(pAVLTreeNode^);
	RecursiveInsert := pAVLTreeNode^;
	RETURN;
END_IF

IF (Key < Node.Key) THEN
	Node.left := THIS^.RecursiveInsert(Key, Value, Node.left);
ELSIF (Key > Node.Key) THEN
	Node.right := THIS^.RecursiveInsert(Key, Value, Node.right);
ELSE
	Node.Reinitialize(Key,Value);
	RecursiveInsert := Node;
END_IF

THIS^.updateHeight(node);

balanceFactor := THIS^.GetBalanceFactor(Node);
Node := balance(Node);
RecursiveInsert := Node;
END_METHOD

METHOD PUBLIC Remove
VAR_INPUT
	Key : T_MAXSTRING;
END_VAR
rootNode := THIS^.RecursiveDelete(Key, rootNode);
EmitChangedEvent();
END_METHOD

METHOD PRIVATE RemoveNode
VAR_INPUT
	Node : I_OrderedDictionaryTreeNode;
END_VAR
IF Node = head AND Node.Next = 0 THEN
	head := 0;
	tail := 0; 
	RETURN;
END_IF

IF Node = tail AND Node.Previous = 0 THEN
	head := 0;
	tail := 0; 
	RETURN;
END_IF

IF Node = head THEN
	Node.Next.Previous := 0;
	head := Node.Next;
	RETURN;
END_IF

IF Node = tail THEN
	Node.Previous.Next := 0;
	tail := Node.Previous;
	RETURN;
END_IF

// we need to perform this check as replaced nodes may not be head or tail
// but will have had the previous and next removed. Therefore only true deletes
// will have these set.
IF Node.Previous <> 0 AND Node.Next <> 0 THEN
	Node.Previous.Next := Node.Next;
	Node.Next.Previous := Node.Previous;
END_IF
END_METHOD

METHOD PRIVATE ReplaceClonedNodeInOrder
VAR_INPUT
	NodeCloned : I_OrderedDictionaryTreeNode;
	NodeToBeRemoved : I_OrderedDictionaryTreeNode;
END_VAR
IF NodeToBeRemoved = head THEN
	head := NodeCloned;
END_IF

IF NodeToBeRemoved = tail THEN
	tail := NodeCloned;
END_IF

IF NodeCloned.Previous <> 0 THEN
	NodeCloned.Previous.Next := NodeCloned;
END_IF
NodeToBeRemoved.Previous := 0;

IF NodeCloned.Next <> 0 THEN
	NodeCloned.Next.Previous := NodeCloned;
END_IF
NodeToBeRemoved.Next := 0;
END_METHOD

METHOD PRIVATE RightRotate : I_OrderedDictionaryTreeNode
VAR_INPUT
	Y : I_OrderedDictionaryTreeNode;
END_VAR
VAR
	x : I_OrderedDictionaryTreeNode;
	t2 : I_OrderedDictionaryTreeNode;
END_VAR
x := Y.left;
t2 := x.right;
x.right := Y;
Y.left := t2;
THIS^.UpdateHeight(Y);
THIS^.UpdateHeight(x);
RightRotate := x;
END_METHOD

METHOD PUBLIC TryAdd : BOOL
VAR_INPUT
	Key : T_MAXSTRING;
	Value : ANY;
END_VAR
IF ContainsKey(Key) THEN
	RETURN;
END_IF
	  
THIS^.AddOrUpdate(Key, Value);
TryAdd := TRUE;
END_METHOD

METHOD PUBLIC TryGetValue : BOOL
VAR_INPUT
	Key : T_MAXSTRING;
	Destination	: ANY;
END_VAR
TryGetValue := TryGetValueTo(Key, Destination.pValue, DINT_TO_UDINT(Destination.diSize));
END_METHOD

METHOD PUBLIC TryGetValueTo : BOOL
VAR_INPUT
	Key : T_MAXSTRING;
	DestinationAddress : PVOID;
	DestinationSize : UDINT;
END_VAR
VAR
	foundNode : I_OrderedDictionaryTreeNode;
END_VAR
foundNode := THIS^.RecursiveFind(Key, rootNode);

IF foundNode = 0 THEN
	RETURN;
END_IF

TryGetValueTo := foundNode.TryGetTo(DestinationAddress, DestinationSize);
END_METHOD

METHOD PRIVATE UpdateHeight
VAR_INPUT
	Node : I_OrderedDictionaryTreeNode;
END_VAR
IF (Node = 0) THEN
	RETURN;
END_IF

Node.height := 1 + MAX(THIS^.GetHeight(Node.left), THIS^.GetHeight(Node.right));
END_METHOD

END_FUNCTION_BLOCK

// ---- _Internal/OrderedDictionary/Enumerator/OrderedDictionaryForwardEnumerator.TcPOU
{attribute 'linkalways'} 
{attribute 'no_explicit_call' := 'This FB is a CLASS and must be accessed using methods or properties'}
{attribute 'enable_dynamic_creation'}
FUNCTION_BLOCK OrderedDictionaryForwardEnumerator EXTENDS Disposable IMPLEMENTS I_KeyValueForwardEnumerator, I_EventHandler
VAR
	parent : I_Dictionary;
	nodes : I_Collection;
	collectionEnumerator : I_ForwardEnumerator;
	currentNode : I_OrderedDictionaryTreeNode;
	moveNextCalled : BOOL := FALSE;
	invalid : BOOL := FALSE; 
END_VAR

METHOD FB_exit : BOOL
VAR_INPUT
	bInCopyCode : BOOL; // if TRUE, the exit method is called for exiting an instance that is copied afterwards (online change).
END_VAR
IF bInCopyCode THEN
	RETURN;
END_IF

collectionEnumerator.Dispose();
nodes.Dispose();

IF parent = 0 THEN
	RETURN;
END_IF

parent.OffEvent('OnChanged',THIS^);
parent.OffEvent('OnDisposed',THIS^);
END_METHOD

METHOD FB_init : BOOL
VAR_INPUT
	bInitRetains : BOOL; // if TRUE, the retain variables are initialized (warm start / cold start)
	bInCopyCode : BOOL;  // if TRUE, the instance afterwards gets moved into the copy code (online change)
	Parent : I_Dictionary;
	Nodes : I_Collection;
END_VAR
Parent.OnEvent('OnChanged',THIS^);
Parent.OnEvent('OnDisposed',THIS^);
THIS^.parent := Parent;
THIS^.nodes := Nodes;
THIS^.collectionEnumerator := Nodes.GetEnumerator();
END_METHOD

METHOD PUBLIC HandleEvent
VAR_INPUT
	Event : I_Event;
END_VAR
VAR
	changedEvent : I_KeyValueCollectionChangedEvent;
	disposedEvent : I_KeyValueCollectionDisposedEvent;
END_VAR
IF __QUERYINTERFACE(Event, changedEvent) THEN
	invalid := TRUE;
	currentNode := 0;
ELSIF __QUERYINTERFACE(Event, disposedEvent) THEN
	parent := 0;	
	Dispose();
END_IF
END_METHOD

PROPERTY PUBLIC IsValid : BOOL
GET // PUBLIC
IsValid := (not invalid and parent <> 0);
END_GET
END_PROPERTY

PROPERTY PUBLIC Key : T_MAXSTRING
GET
IF NOT IsValid THEN
	RETURN;
END_IF

IF currentNode = 0 THEN
	RETURN;
END_IF

Key := currentNode.Key;
END_GET
END_PROPERTY

METHOD PUBLIC MoveNext : BOOL
IF invalid THEN
	RETURN;
END_IF

IF collectionEnumerator.MoveNext() THEN
	collectionEnumerator.TryGet(currentNode);
	MoveNext := TRUE;
END_IF
END_METHOD

METHOD Reset
VAR_INPUT
END_VAR
moveNextCalled := FALSE;
collectionEnumerator.Reset();
END_METHOD

METHOD PUBLIC TryGet : BOOL;
VAR_INPUT
	Destination : ANY;
END_VAR
IF currentNode <> 0 THEN
	TryGet := currentNode.TryGet(Destination);
END_IF
END_METHOD

METHOD PUBLIC TryGetTo : BOOL;
VAR_INPUT
	DestinationAddress : PVOID;
	DestinationSize : UDINT;
END_VAR
IF currentNode <> 0 THEN
	TryGetTo := currentNode.TryGetTo(DestinationAddress,DestinationSize);
END_IF
END_METHOD

END_FUNCTION_BLOCK

// ---- _Internal/OrderedDictionary/Node/OrderedDictionaryTreeNode.TcPOU
{attribute 'linkalways'} 
{attribute 'no_explicit_call' := 'This FB is a CLASS and must be accessed using methods or properties'}
{attribute 'enable_dynamic_creation'}
FUNCTION_BLOCK OrderedDictionaryTreeNode EXTENDS Disposable IMPLEMENTS I_OrderedDictionaryTreeNode
VAR
	_key : T_MAXSTRING;
	pBuffer : POINTER TO BYTE;
	bufferSize : UDINT;
    _height : DINT;
    _left : I_OrderedDictionaryTreeNode;
    _right : I_OrderedDictionaryTreeNode;
	_next : I_OrderedDictionaryTreeNode;
    _previous : I_OrderedDictionaryTreeNode;
END_VAR

METHOD PUBLIC Clone
VAR_INPUT
	Node : I_OrderedDictionaryTreeNode;
END_VAR
DestroyBuffer();
CreateBuffer(Node.NodeBufferSize);
CopySourceToBuffer(Node.NodeBufferPointer);
_key := Node.Key;
_previous := Node.Previous;
_next := Node.Next;
END_METHOD

METHOD PRIVATE CopyBufferToDestination
VAR_INPUT
	DestinationAddress : PVOID;
END_VAR
MEMCPY(DestinationAddress, pBuffer, bufferSize);
END_METHOD

METHOD PRIVATE CopySourceToBuffer
VAR_INPUT
	SourceAddress : PVOID;
END_VAR
MEMCPY(pBuffer, SourceAddress, bufferSize);
END_METHOD

METHOD PRIVATE CreateBuffer
VAR_INPUT
	SizeInBytes : UDINT;
END_VAR
bufferSize := SizeInBytes;
pBuffer := __NEW(BYTE, SizeInBytes);
END_METHOD

PROPERTY PUBLIC DataSize : UDINT
GET
DataSize := bufferSize;
END_GET
END_PROPERTY

METHOD PRIVATE DestroyBuffer
VAR_INPUT
END_VAR
IF pBuffer = 0 THEN
	RETURN;
END_IF

__DELETE(pBuffer);
bufferSize := 0;
END_METHOD

METHOD PUBLIC Equals : BOOL
VAR_INPUT
	Symbol : ANY;
END_VAR
IF pBuffer = 0 THEN
	RETURN;
END_IF

IF bufferSize <> DINT_TO_UDINT(symbol.diSize) THEN
	RETURN;
END_IF

Equals := MEMCMP(Symbol.pValue, pBuffer, bufferSize) = 0;
END_METHOD

METHOD FB_exit : BOOL
VAR_INPUT
	bInCopyCode : BOOL; // if TRUE, the exit method is called for exiting an instance that is copied afterwards (online change).
END_VAR
IF bInCopyCode THEN
	RETURN;
END_IF

DestroyBuffer();
END_METHOD

METHOD FB_init : BOOL
VAR_INPUT
	bInitRetains : BOOL; // if TRUE, the retain variables are initialized (warm start / cold start)
	bInCopyCode : BOOL;  // if TRUE, the instance afterwards gets moved into the copy code (online change)
	NodeKey : T_MAXSTRING;
	NodeSource : ANY;
END_VAR
_key := NodeKey;
CreateBuffer(DINT_TO_UDINT(NodeSource.diSize));
CopySourceToBuffer(NodeSource.pValue);
END_METHOD

PROPERTY PUBLIC Height : DINT
GET
Height := _height;
END_GET
SET // PUBLIC
_height := Height;
END_SET
END_PROPERTY

PROPERTY PUBLIC Key : T_MAXSTRING
GET
Key := _key;
END_GET
END_PROPERTY

PROPERTY PUBLIC Left : I_OrderedDictionaryTreeNode
GET
Left := _left;
END_GET
SET
_left := Left;
END_SET
END_PROPERTY

PROPERTY PUBLIC Next : I_OrderedDictionaryTreeNode
GET
Next := _next;
END_GET
SET
_next := Next;
END_SET
END_PROPERTY

PROPERTY PUBLIC NodeBufferPointer : Pointer To Byte
GET
NodeBufferPointer := pBuffer;
END_GET
END_PROPERTY

PROPERTY PUBLIC NodeBufferSize : UDINT
GET
NodeBufferSize := bufferSize;
END_GET
END_PROPERTY

PROPERTY PUBLIC Previous : I_OrderedDictionaryTreeNode
GET
Previous := _previous;
END_GET
SET
_previous := Previous;
END_SET
END_PROPERTY

METHOD Reinitialize
VAR_INPUT
	Key : T_MAXSTRING;
	Source : ANY;
END_VAR
_key := Key;

IF pBuffer <> 0 THEN
	DestroyBuffer();
END_IF

CreateBuffer(DINT_TO_UDINT(Source.diSize));
CopySourceToBuffer(Source.pValue);
END_METHOD

PROPERTY PUBLIC Right : I_OrderedDictionaryTreeNode
GET
Right := _right;
END_GET
SET
_right := Right;
END_SET
END_PROPERTY

METHOD TryGet : BOOL
VAR_INPUT
	Destination	: ANY;
END_VAR
TryGet := TryGetTo(Destination.pValue, DINT_TO_UDINT(Destination.diSize));
END_METHOD

METHOD TryGetTo : BOOL
VAR_INPUT
	DestinationAddress : PVOID;
	DestinationSize : UDINT;
END_VAR
IF pBuffer = 0 THEN
	RETURN;
END_IF

IF bufferSize <> DestinationSize THEN
	RETURN;
END_IF

CopyBufferToDestination(DestinationAddress);
TryGetTo := TRUE;
END_METHOD

END_FUNCTION_BLOCK

// ---- Queue/Queue.TcPOU
{attribute 'linkalways'} 
{attribute 'no_explicit_call' := 'This FB is a CLASS and must be accessed using methods or properties'}
{attribute 'enable_dynamic_creation'}
FUNCTION_BLOCK Queue EXTENDS Disposable IMPLEMENTS I_Queue
VAR
	linkedList : LinkedList;
	eventEmitter : EventEmitter;
END_VAR

METHOD PUBLIC AddItem
VAR_INPUT
	Item : ANY;
END_VAR
Enqueue(Item);
END_METHOD

METHOD PUBLIC Clear
linkedList.Clear();
EmitChangedEvent();
END_METHOD

METHOD PUBLIC Contains : BOOL;
VAR_INPUT
	Item : ANY;
END_VAR
VAR
	found : I_LinkedListNode;
END_VAR
found := linkedList.Find(Item);
Contains := found <> 0;
END_METHOD

PROPERTY PUBLIC Count : DINT
GET
Count := linkedList.Count;
END_GET
END_PROPERTY

METHOD PRIVATE EmitChangedEvent
VAR
	pCollectionChangedEvent : POINTER TO CollectionChangedEvent;
END_VAR
pCollectionChangedEvent := __NEW(CollectionChangedEvent(Target := THIS^));
eventEmitter.Emit('OnChanged', pCollectionChangedEvent^);
pCollectionChangedEvent^.Dispose();
END_METHOD

METHOD PRIVATE EmitDisposedEvent
VAR
	pCollectionDisposedEvent : POINTER TO CollectionDisposedEvent;
END_VAR
pCollectionDisposedEvent := __NEW(CollectionDisposedEvent(Target := THIS^));
eventEmitter.Emit('OnDisposed', pCollectionDisposedEvent^);
pCollectionDisposedEvent^.Dispose();
END_METHOD

METHOD PUBLIC Enqueue
VAR_INPUT
	Item : ANY;
END_VAR
linkedList.AddLast(Item);
EmitChangedEvent();
END_METHOD

METHOD FB_exit : BOOL
VAR_INPUT
	bInCopyCode : BOOL; // if TRUE, the exit method is called for exiting an instance that is copied afterwards (online change).
END_VAR
IF bInCopyCode THEN
	RETURN;
END_IF

Clear();
EmitDisposedEvent();
END_METHOD

METHOD PUBLIC GetEnumerator : I_ForwardEnumerator
GetEnumerator := linkedList.GetEnumerator();
END_METHOD

PROPERTY IsEmpty : BOOL
GET
IsEmpty := linkedList.IsEmpty;
END_GET
END_PROPERTY

METHOD PUBLIC OffEvent
VAR_INPUT
	EventName : T_MaxString;
	EventHandler : I_EventHandler;
END_VAR
eventEmitter.OffEvent(EventName, EventHandler);
END_METHOD

METHOD PUBLIC OnceEvent
VAR_INPUT
	EventName : T_MaxString;
	EventHandler : I_EventHandler;
END_VAR
eventEmitter.OnceEvent(EventName, EventHandler);
END_METHOD

METHOD PUBLIC OnEvent
VAR_INPUT
	EventName : T_MaxString;
	EventHandler : I_EventHandler;
END_VAR
eventEmitter.OnEvent(EventName, EventHandler);
END_METHOD

METHOD PUBLIC TryCopyTo : BOOL
VAR_INPUT
	Destination : ANY;
END_VAR
TryCopyTo := linkedList.TryCopyTo(Destination);
END_METHOD

METHOD PUBLIC TryCopyToLocation : BOOL
VAR_INPUT
	DestinationAddress : PVOID;
	DestinationSize : UDINT;
END_VAR
TryCopyToLocation := linkedList.TryCopyToLocation(DestinationAddress, DestinationSize);
END_METHOD

METHOD PUBLIC TryDequeue : BOOL;
VAR_INPUT
	Destination : ANY;
END_VAR
VAR
	first : I_LinkedListNode;
	dequeued : BOOL;
END_VAR
first := linkedList.First;

IF first = 0 THEN
	RETURN;
END_IF

dequeued := linkedList.First.TryGet(Destination);

IF NOT dequeued THEN
	RETURN;
END_IF

linkedList.RemoveFirst();
EmitChangedEvent();
TryDequeue := TRUE;
END_METHOD

METHOD PUBLIC TryPeek : BOOL;
VAR_INPUT
	Destination : ANY;
END_VAR
VAR
	first : I_LinkedListNode;
END_VAR
first := linkedList.First;

IF first = 0 THEN
	RETURN;
END_IF

TryPeek := first.TryGet(Destination);
END_METHOD

METHOD PUBLIC TryRemoveItem : BOOL
VAR_INPUT
	Item : ANY;
END_VAR
TryRemoveItem := linkedList.TryRemoveItem(Item);
EmitChangedEvent();
END_METHOD

END_FUNCTION_BLOCK

// ---- Stack/Stack.TcPOU
{attribute 'linkalways'} 
{attribute 'no_explicit_call' := 'This FB is a CLASS and must be accessed using methods or properties'}
{attribute 'enable_dynamic_creation'}
FUNCTION_BLOCK Stack EXTENDS Disposable IMPLEMENTS I_Stack
VAR
	linkedList : LinkedList;
	eventEmitter : EventEmitter;
END_VAR

METHOD PUBLIC AddItem
VAR_INPUT
	Item : ANY;
END_VAR
Push(Item);
END_METHOD

METHOD PUBLIC Clear
linkedList.Clear();
EmitChangedEvent();
END_METHOD

METHOD PUBLIC Contains : BOOL;
VAR_INPUT
	Item : ANY;
END_VAR
VAR
	found : I_LinkedListNode;
END_VAR
found := linkedList.Find(Item);
Contains := found <> 0;
END_METHOD

PROPERTY PUBLIC Count : DINT
GET
Count := linkedList.Count;
END_GET
END_PROPERTY

METHOD PRIVATE EmitChangedEvent
VAR
	pCollectionChangedEvent : POINTER TO CollectionChangedEvent;
END_VAR
pCollectionChangedEvent := __NEW(CollectionChangedEvent(Target := THIS^));
eventEmitter.Emit('OnChanged', pCollectionChangedEvent^);
pCollectionChangedEvent^.Dispose();
END_METHOD

METHOD PRIVATE EmitDisposedEvent
VAR
	pCollectionDisposedEvent : POINTER TO CollectionDisposedEvent;
END_VAR
pCollectionDisposedEvent := __NEW(CollectionDisposedEvent(Target := THIS^));
eventEmitter.Emit('OnDisposed', pCollectionDisposedEvent^);
pCollectionDisposedEvent^.Dispose();
END_METHOD

METHOD FB_exit : BOOL
VAR_INPUT
	bInCopyCode : BOOL; // if TRUE, the exit method is called for exiting an instance that is copied afterwards (online change).
END_VAR
IF bInCopyCode THEN
	RETURN;
END_IF

Clear();
EmitDisposedEvent();
END_METHOD

METHOD PUBLIC GetEnumerator : I_ForwardEnumerator
GetEnumerator := linkedList.GetEnumerator();
END_METHOD

PROPERTY IsEmpty : BOOL
GET
IsEmpty := linkedList.IsEmpty;
END_GET
END_PROPERTY

METHOD PUBLIC OffEvent
VAR_INPUT
	EventName : T_MaxString;
	EventHandler : I_EventHandler;
END_VAR
eventEmitter.OffEvent(EventName, EventHandler);
END_METHOD

METHOD PUBLIC OnceEvent
VAR_INPUT
	EventName : T_MaxString;
	EventHandler : I_EventHandler;
END_VAR
eventEmitter.OnceEvent(EventName, EventHandler);
END_METHOD

METHOD PUBLIC OnEvent
VAR_INPUT
	EventName : T_MaxString;
	EventHandler : I_EventHandler;
END_VAR
eventEmitter.OnEvent(EventName, EventHandler);
END_METHOD

METHOD PUBLIC Push
VAR_INPUT
	Item : ANY;
END_VAR
linkedList.AddFirst(Item);
EmitChangedEvent();
END_METHOD

METHOD PUBLIC TryCopyTo : BOOL
VAR_INPUT
	Destination : ANY;
END_VAR
TryCopyTo := linkedList.TryCopyTo(Destination);
END_METHOD

METHOD PUBLIC TryCopyToLocation : BOOL
VAR_INPUT
	DestinationAddress : PVOID;
	DestinationSize : UDINT;
END_VAR
TryCopyToLocation := linkedList.TryCopyToLocation(DestinationAddress, DestinationSize);
END_METHOD

METHOD PUBLIC TryPeek : BOOL;
VAR_INPUT
	Destination : ANY;
END_VAR
VAR
	first : I_LinkedListNode;
END_VAR
first := linkedList.First;

IF first = 0 THEN
	RETURN;
END_IF

TryPeek := first.TryGet(Destination);
END_METHOD

METHOD PUBLIC TryPop : BOOL;
VAR_INPUT
	Destination : ANY;
END_VAR
VAR
	first : I_LinkedListNode;
	popped : BOOL;
END_VAR
first := linkedList.First;

IF first = 0 THEN
	RETURN;
END_IF

popped := linkedList.First.TryGet(Destination);

IF NOT popped THEN
	RETURN;
END_IF

linkedList.RemoveFirst();
EmitChangedEvent();
TryPop := TRUE;
END_METHOD

METHOD PUBLIC TryRemoveItem : BOOL
VAR_INPUT
	Item : ANY;
END_VAR
TryRemoveItem := linkedList.TryRemoveItem(Item);
EmitChangedEvent();
END_METHOD

END_FUNCTION_BLOCK
